KUKA KRL data list: profile_defaut.dat

&ACCESS RVP
&PARAM EDITMASK = *
DEFDAT  profile_defaut
;FOLD EXTERNAL DECLARATIONS;%{PE}%MKUKATPBASIS,%CEXT,%VCOMMON,%P
;FOLD BASISTECH EXT;%{PE}%MKUKATPBASIS,%CEXT,%VEXT,%P
EXT  BAS (BAS_COMMAND  :IN,REAL  :IN )
DECL INT SUCCESS
;ENDFOLD (BASISTECH EXT)
;FOLD USER EXT;%{E}%MKUKATPUSER,%CEXT,%VEXT,%P
;Make your modifications here

;ENDFOLD (USER EXT)
;ENDFOLD (EXTERNAL DECLARATIONS)

INT APP_GENNUMBER = 215375
INT APP_ANSWER
INT APP_OFFSET
DECL STATE_T APP_STATE

DECL PDAT PPDATP0={VEL 100,ACC 100,APO_DIST 5,APO_MODE #CDIS,GEAR_JERK 100.0,EXAX_IGN 0}
DECL FDAT FP0={TOOL_NO 2,BASE_NO 10,IPO_FRAME #BASE,POINT2[] " ",TQ_STATE FALSE}
DECL E6AXIS XP0={A1 -1000.000,A2 -90.000,A3 90.000,A4 0.000,A5 -90.000,A6 0.000,E1 0.000,E2 0.000,E3 0.000,E4 0.000,E5 0.000,E6 0.000}

; Data for Routine_0
DECL LDAT LCPDATP1={VEL 0.1,ACC 100,APO_DIST 5,APO_FAC 50.0,ORI_TYP #VAR,CIRC_TYP #BASE,JERK_FAC 50.0}
DECL FDAT FP1={TOOL_NO 2,BASE_NO 10,IPO_FRAME #BASE,POINT2[] " ",TQ_STATE FALSE}
DECL E6POS XP1={X -118.780,Y -0.350,Z 2.610,A -0.040,B -12.450,C -29.720}
DECL LDAT LCPDATC2={VEL 0.1,ACC 100,APO_DIST 5,APO_FAC 50.0,ORI_TYP #VAR,CIRC_TYP #BASE,JERK_FAC 50.0}
DECL FDAT FC2={TOOL_NO 2,BASE_NO 10,IPO_FRAME #BASE,POINT2[] " ",TQ_STATE FALSE}
DECL E6POS XCAux2={X -55.000,Y 13.210,Z 2.610,A 0.000,B 0.000,C -32.000}
DECL E6POS XCDes2={X 8.780,Y -0.350,Z 2.610,A 0.040,B 12.450,C -29.720}
DECL LDAT LCPDATC3={VEL 0.5,ACC 100,APO_DIST 5,APO_FAC 50.0,ORI_TYP #VAR,CIRC_TYP #BASE,JERK_FAC 50.0}
DECL FDAT FC3={TOOL_NO 2,BASE_NO 10,IPO_FRAME #BASE,POINT2[] " ",TQ_STATE FALSE}
DECL E6POS XCAux3={X 32.690,Y -13.600,Z 2.610,A 0.100,B 17.240,C -27.390}
DECL E6POS XCDes3={X 31.690,Y -15.080,Z 3.460,A 0.010,B 10.280,C -15.600}
DECL LDAT LCPDATP4={VEL 0.1,ACC 100,APO_DIST 5,APO_FAC 50.0,ORI_TYP #VAR,CIRC_TYP #BASE,JERK_FAC 50.0}
DECL FDAT FP4={TOOL_NO 2,BASE_NO 10,IPO_FRAME #BASE,POINT2[] " ",TQ_STATE FALSE}
DECL E6POS XP4={X 8.050,Y -1.980,Z 3.460,A 0.000,B 7.460,C -17.100}
DECL LDAT LCPDATC5={VEL 0.1,ACC 100,APO_DIST 5,APO_FAC 50.0,ORI_TYP #VAR,CIRC_TYP #BASE,JERK_FAC 50.0}
DECL FDAT FC5={TOOL_NO 2,BASE_NO 10,IPO_FRAME #BASE,POINT2[] " ",TQ_STATE FALSE}
DECL E6POS XCAux5={X -55.000,Y 11.430,Z 3.460,A 0.000,B 0.000,C -18.620}
DECL E6POS XCDes5={X -118.050,Y -1.980,Z 3.460,A -0.000,B -7.460,C -17.100}
DECL LDAT LCPDATC6={VEL 0.5,ACC 100,APO_DIST 5,APO_FAC 50.0,ORI_TYP #VAR,CIRC_TYP #BASE,JERK_FAC 50.0}
DECL FDAT FC6={TOOL_NO 2,BASE_NO 10,IPO_FRAME #BASE,POINT2[] " ",TQ_STATE FALSE}
DECL E6POS XCAux6={X -141.690,Y -15.080,Z 3.460,A -0.010,B -10.280,C -15.600}
DECL E6POS XCDes6={X -140.610,Y -16.680,Z 3.860,A -0.000,B -2.920,C -4.340}
DECL LDAT LCPDATP7={VEL 0.1,ACC 100,APO_DIST 5,APO_FAC 50.0,ORI_TYP #VAR,CIRC_TYP #BASE,JERK_FAC 50.0}
DECL FDAT FP7={TOOL_NO 2,BASE_NO 10,IPO_FRAME #BASE,POINT2[] " ",TQ_STATE FALSE}
DECL E6POS XP7={X -117.270,Y -3.740,Z 3.860,A -0.000,B -2.130,C -4.780}
DECL LDAT LCPDATC8={VEL 0.1,ACC 100,APO_DIST 5,APO_FAC 50.0,ORI_TYP #VAR,CIRC_TYP #BASE,JERK_FAC 50.0}
DECL FDAT FC8={TOOL_NO 2,BASE_NO 10,IPO_FRAME #BASE,POINT2[] " ",TQ_STATE FALSE}
DECL E6POS XCAux8={X -55.000,Y 9.500,Z 3.860,A 0.000,B 0.000,C -5.230}
DECL E6POS XCDes8={X 7.270,Y -3.740,Z 3.860,A 0.000,B 2.130,C -4.780}
DECL LDAT LCPDATC9={VEL 0.5,ACC 100,APO_DIST 5,APO_FAC 50.0,ORI_TYP #VAR,CIRC_TYP #BASE,JERK_FAC 50.0}
DECL FDAT FC9={TOOL_NO 2,BASE_NO 10,IPO_FRAME #BASE,POINT2[] " ",TQ_STATE FALSE}
DECL E6POS XCAux9={X 30.610,Y -16.680,Z 3.860,A 0.000,B 2.920,C -4.340}
DECL E6POS XCDes9={X 30.620,Y -16.670,Z 3.900,A 0.000,B 0.000,C -0.000}
DECL LDAT LCPDATP10={VEL 0.1,ACC 100,APO_DIST 5,APO_FAC 50.0,ORI_TYP #VAR,CIRC_TYP #BASE,JERK_FAC 50.0}
DECL FDAT FP10={TOOL_NO 2,BASE_NO 10,IPO_FRAME #BASE,POINT2[] " ",TQ_STATE FALSE}
DECL E6POS XP10={X 7.270,Y -3.730,Z 3.900,A 0.000,B 0.000,C -0.000}
DECL LDAT LCPDATC11={VEL 0.1,ACC 100,APO_DIST 5,APO_FAC 50.0,ORI_TYP #VAR,CIRC_TYP #BASE,JERK_FAC 50.0}
DECL FDAT FC11={TOOL_NO 2,BASE_NO 10,IPO_FRAME #BASE,POINT2[] " ",TQ_STATE FALSE}
DECL E6POS XCAux11={X -55.000,Y 9.510,Z 3.900,A 0.000,B 0.000,C -0.000}
DECL E6POS XCDes11={X -117.270,Y -3.730,Z 3.900,A 0.000,B 0.000,C -0.000}
DECL LDAT LCPDATC12={VEL 0.5,ACC 100,APO_DIST 5,APO_FAC 50.0,ORI_TYP #VAR,CIRC_TYP #BASE,JERK_FAC 50.0}
DECL FDAT FC12={TOOL_NO 2,BASE_NO 10,IPO_FRAME #BASE,POINT2[] " ",TQ_STATE FALSE}
DECL E6POS XCAux12={X -140.620,Y -16.670,Z 3.900,A 0.000,B 0.000,C -0.000}
DECL E6POS XCDes12={X -139.500,Y -18.330,Z 3.900,A 0.000,B 0.000,C -0.000}
DECL LDAT LCPDATP13={VEL 0.1,ACC 100,APO_DIST 5,APO_FAC 50.0,ORI_TYP #VAR,CIRC_TYP #BASE,JERK_FAC 50.0}
DECL FDAT FP13={TOOL_NO 2,BASE_NO 10,IPO_FRAME #BASE,POINT2[] " ",TQ_STATE FALSE}
DECL E6POS XP13={X -116.460,Y -5.560,Z 3.900,A 0.000,B 0.000,C -0.000}
DECL LDAT LCPDATC14={VEL 0.1,ACC 100,APO_DIST 5,APO_FAC 50.0,ORI_TYP #VAR,CIRC_TYP #BASE,JERK_FAC 50.0}
DECL FDAT FC14={TOOL_NO 2,BASE_NO 10,IPO_FRAME #BASE,POINT2[] " ",TQ_STATE FALSE}
DECL E6POS XCAux14={X -55.000,Y 7.510,Z 3.900,A 0.000,B 0.000,C -0.000}
DECL E6POS XCDes14={X 6.460,Y -5.560,Z 3.900,A 0.000,B 0.000,C -0.000}
DECL LDAT LCPDATC15={VEL 0.5,ACC 100,APO_DIST 5,APO_FAC 50.0,ORI_TYP #VAR,CIRC_TYP #BASE,JERK_FAC 50.0}
DECL FDAT FC15={TOOL_NO 2,BASE_NO 10,IPO_FRAME #BASE,POINT2[] " ",TQ_STATE FALSE}
DECL E6POS XCAux15={X 29.500,Y -18.330,Z 3.900,A 0.000,B 0.000,C -0.000}
DECL E6POS XCDes15={X 28.380,Y -19.990,Z 3.900,A 0.000,B 0.000,C -0.000}
DECL LDAT LCPDATP16={VEL 0.1,ACC 100,APO_DIST 5,APO_FAC 50.0,ORI_TYP #VAR,CIRC_TYP #BASE,JERK_FAC 50.0}
DECL FDAT FP16={TOOL_NO 2,BASE_NO 10,IPO_FRAME #BASE,POINT2[] " ",TQ_STATE FALSE}
DECL E6POS XP16={X 5.650,Y -7.390,Z 3.900,A 0.000,B 0.000,C -0.000}
DECL LDAT LCPDATC17={VEL 0.1,ACC 100,APO_DIST 5,APO_FAC 50.0,ORI_TYP #VAR,CIRC_TYP #BASE,JERK_FAC 50.0}
DECL FDAT FC17={TOOL_NO 2,BASE_NO 10,IPO_FRAME #BASE,POINT2[] " ",TQ_STATE FALSE}
DECL E6POS XCAux17={X -55.000,Y 5.510,Z 3.900,A 0.000,B 0.000,C -0.000}
DECL E6POS XCDes17={X -115.650,Y -7.390,Z 3.900,A 0.000,B 0.000,C -0.000}
DECL LDAT LCPDATC18={VEL 0.5,ACC 100,APO_DIST 5,APO_FAC 50.0,ORI_TYP #VAR,CIRC_TYP #BASE,JERK_FAC 50.0}
DECL FDAT FC18={TOOL_NO 2,BASE_NO 10,IPO_FRAME #BASE,POINT2[] " ",TQ_STATE FALSE}
DECL E6POS XCAux18={X -138.380,Y -19.990,Z 3.900,A 0.000,B 0.000,C -0.000}
DECL E6POS XCDes18={X -137.260,Y -21.640,Z 3.900,A 0.000,B 0.000,C -0.000}
DECL LDAT LCPDATP19={VEL 0.1,ACC 100,APO_DIST 5,APO_FAC 50.0,ORI_TYP #VAR,CIRC_TYP #BASE,JERK_FAC 50.0}
DECL FDAT FP19={TOOL_NO 2,BASE_NO 10,IPO_FRAME #BASE,POINT2[] " ",TQ_STATE FALSE}
DECL E6POS XP19={X -114.830,Y -9.210,Z 3.900,A 0.000,B 0.000,C -0.000}
DECL LDAT LCPDATC20={VEL 0.1,ACC 100,APO_DIST 5,APO_FAC 50.0,ORI_TYP #VAR,CIRC_TYP #BASE,JERK_FAC 50.0}
DECL FDAT FC20={TOOL_NO 2,BASE_NO 10,IPO_FRAME #BASE,POINT2[] " ",TQ_STATE FALSE}
DECL E6POS XCAux20={X -55.000,Y 3.510,Z 3.900,A 0.000,B 0.000,C -0.000}
DECL E6POS XCDes20={X 4.830,Y -9.210,Z 3.900,A 0.000,B 0.000,C -0.000}
DECL LDAT LCPDATC21={VEL 0.5,ACC 100,APO_DIST 5,APO_FAC 50.0,ORI_TYP #VAR,CIRC_TYP #BASE,JERK_FAC 50.0}
DECL FDAT FC21={TOOL_NO 2,BASE_NO 10,IPO_FRAME #BASE,POINT2[] " ",TQ_STATE FALSE}
DECL E6POS XCAux21={X 27.260,Y -21.640,Z 3.900,A 0.000,B 0.000,C -0.000}
DECL E6POS XCDes21={X 26.140,Y -23.300,Z 3.900,A 0.000,B 0.000,C -0.000}
DECL LDAT LCPDATP22={VEL 0.1,ACC 100,APO_DIST 5,APO_FAC 50.0,ORI_TYP #VAR,CIRC_TYP #BASE,JERK_FAC 50.0}
DECL FDAT FP22={TOOL_NO 2,BASE_NO 10,IPO_FRAME #BASE,POINT2[] " ",TQ_STATE FALSE}
DECL E6POS XP22={X 4.020,Y -11.040,Z 3.900,A 0.000,B 0.000,C -0.000}
DECL LDAT LCPDATC23={VEL 0.1,ACC 100,APO_DIST 5,APO_FAC 50.0,ORI_TYP #VAR,CIRC_TYP #BASE,JERK_FAC 50.0}
DECL FDAT FC23={TOOL_NO 2,BASE_NO 10,IPO_FRAME #BASE,POINT2[] " ",TQ_STATE FALSE}
DECL E6POS XCAux23={X -55.000,Y 1.510,Z 3.900,A 0.000,B 0.000,C -0.000}
DECL E6POS XCDes23={X -114.020,Y -11.040,Z 3.900,A 0.000,B 0.000,C -0.000}
DECL LDAT LCPDATC24={VEL 0.5,ACC 100,APO_DIST 5,APO_FAC 50.0,ORI_TYP #VAR,CIRC_TYP #BASE,JERK_FAC 50.0}
DECL FDAT FC24={TOOL_NO 2,BASE_NO 10,IPO_FRAME #BASE,POINT2[] " ",TQ_STATE FALSE}
DECL E6POS XCAux24={X -136.140,Y -23.300,Z 3.900,A 0.000,B 0.000,C -0.000}
DECL E6POS XCDes24={X -135.020,Y -24.960,Z 3.900,A 0.000,B 0.000,C -0.000}
DECL LDAT LCPDATP25={VEL 0.1,ACC 100,APO_DIST 5,APO_FAC 50.0,ORI_TYP #VAR,CIRC_TYP #BASE,JERK_FAC 50.0}
DECL FDAT FP25={TOOL_NO 2,BASE_NO 10,IPO_FRAME #BASE,POINT2[] " ",TQ_STATE FALSE}
DECL E6POS XP25={X -113.210,Y -12.870,Z 3.900,A 0.000,B 0.000,C -0.000}
DECL LDAT LCPDATC26={VEL 0.1,ACC 100,APO_DIST 5,APO_FAC 50.0,ORI_TYP #VAR,CIRC_TYP #BASE,JERK_FAC 50.0}
DECL FDAT FC26={TOOL_NO 2,BASE_NO 10,IPO_FRAME #BASE,POINT2[] " ",TQ_STATE FALSE}
DECL E6POS XCAux26={X -55.000,Y -0.490,Z 3.900,A 0.000,B 0.000,C -0.000}
DECL E6POS XCDes26={X 3.210,Y -12.870,Z 3.900,A 0.000,B 0.000,C -0.000}
DECL LDAT LCPDATC27={VEL 0.5,ACC 100,APO_DIST 5,APO_FAC 50.0,ORI_TYP #VAR,CIRC_TYP #BASE,JERK_FAC 50.0}
DECL FDAT FC27={TOOL_NO 2,BASE_NO 10,IPO_FRAME #BASE,POINT2[] " ",TQ_STATE FALSE}
DECL E6POS XCAux27={X 25.020,Y -24.960,Z 3.900,A 0.000,B 0.000,C -0.000}
DECL E6POS XCDes27={X 23.910,Y -26.620,Z 3.900,A 0.000,B 0.000,C -0.000}
DECL LDAT LCPDATP28={VEL 0.1,ACC 100,APO_DIST 5,APO_FAC 50.0,ORI_TYP #VAR,CIRC_TYP #BASE,JERK_FAC 50.0}
DECL FDAT FP28={TOOL_NO 2,BASE_NO 10,IPO_FRAME #BASE,POINT2[] " ",TQ_STATE FALSE}
DECL E6POS XP28={X 2.390,Y -14.690,Z 3.900,A 0.000,B 0.000,C -0.000}
DECL LDAT LCPDATC29={VEL 0.1,ACC 100,APO_DIST 5,APO_FAC 50.0,ORI_TYP #VAR,CIRC_TYP #BASE,JERK_FAC 50.0}
DECL FDAT FC29={TOOL_NO 2,BASE_NO 10,IPO_FRAME #BASE,POINT2[] " ",TQ_STATE FALSE}
DECL E6POS XCAux29={X -55.000,Y -2.490,Z 3.900,A 0.000,B 0.000,C -0.000}
DECL E6POS XCDes29={X -112.390,Y -14.690,Z 3.900,A 0.000,B 0.000,C -0.000}
DECL LDAT LCPDATC30={VEL 0.5,ACC 100,APO_DIST 5,APO_FAC 50.0,ORI_TYP #VAR,CIRC_TYP #BASE,JERK_FAC 50.0}
DECL FDAT FC30={TOOL_NO 2,BASE_NO 10,IPO_FRAME #BASE,POINT2[] " ",TQ_STATE FALSE}
DECL E6POS XCAux30={X -133.910,Y -26.620,Z 3.900,A 0.000,B 0.000,C -0.000}
DECL E6POS XCDes30={X -132.790,Y -28.280,Z 3.900,A 0.000,B 0.000,C -0.000}
DECL LDAT LCPDATP31={VEL 0.1,ACC 100,APO_DIST 5,APO_FAC 50.0,ORI_TYP #VAR,CIRC_TYP #BASE,JERK_FAC 50.0}
DECL FDAT FP31={TOOL_NO 2,BASE_NO 10,IPO_FRAME #BASE,POINT2[] " ",TQ_STATE FALSE}
DECL E6POS XP31={X -111.580,Y -16.520,Z 3.900,A 0.000,B 0.000,C -0.000}
DECL LDAT LCPDATC32={VEL 0.1,ACC 100,APO_DIST 5,APO_FAC 50.0,ORI_TYP #VAR,CIRC_TYP #BASE,JERK_FAC 50.0}
DECL FDAT FC32={TOOL_NO 2,BASE_NO 10,IPO_FRAME #BASE,POINT2[] " ",TQ_STATE FALSE}
DECL E6POS XCAux32={X -55.000,Y -4.490,Z 3.900,A 0.000,B 0.000,C -0.000}
DECL E6POS XCDes32={X 1.580,Y -16.520,Z 3.900,A 0.000,B 0.000,C -0.000}
DECL LDAT LCPDATC33={VEL 0.5,ACC 100,APO_DIST 5,APO_FAC 50.0,ORI_TYP #VAR,CIRC_TYP #BASE,JERK_FAC 50.0}
DECL FDAT FC33={TOOL_NO 2,BASE_NO 10,IPO_FRAME #BASE,POINT2[] " ",TQ_STATE FALSE}
DECL E6POS XCAux33={X 22.790,Y -28.280,Z 3.900,A 0.000,B 0.000,C -0.000}
DECL E6POS XCDes33={X 22.000,Y -29.440,Z 3.900,A 0.000,B 0.090,C -0.140}
DECL LDAT LCPDATP34={VEL 0.1,ACC 100,APO_DIST 5,APO_FAC 50.0,ORI_TYP #VAR,CIRC_TYP #BASE,JERK_FAC 50.0}
DECL FDAT FP34={TOOL_NO 2,BASE_NO 10,IPO_FRAME #BASE,POINT2[] " ",TQ_STATE FALSE}
DECL E6POS XP34={X 1.010,Y -17.800,Z 3.900,A 0.000,B 0.070,C -0.150}
DECL LDAT LCPDATC35={VEL 0.1,ACC 100,APO_DIST 5,APO_FAC 50.0,ORI_TYP #VAR,CIRC_TYP #BASE,JERK_FAC 50.0}
DECL FDAT FC35={TOOL_NO 2,BASE_NO 10,IPO_FRAME #BASE,POINT2[] " ",TQ_STATE FALSE}
DECL E6POS XCAux35={X -55.000,Y -5.900,Z 3.900,A 0.000,B 0.000,C -0.170}
DECL E6POS XCDes35={X -111.010,Y -17.800,Z 3.900,A -0.000,B -0.070,C -0.150}
DECL LDAT LCPDATC36={VEL 0.5,ACC 100,APO_DIST 5,APO_FAC 50.0,ORI_TYP #VAR,CIRC_TYP #BASE,JERK_FAC 50.0}
DECL FDAT FC36={TOOL_NO 2,BASE_NO 10,IPO_FRAME #BASE,POINT2[] " ",TQ_STATE FALSE}
DECL E6POS XCAux36={X -132.000,Y -29.440,Z 3.900,A -0.000,B -0.090,C -0.140}
DECL E6POS XCDes36={X -130.910,Y -31.070,Z 3.680,A -0.000,B 7.350,C 11.020}
DECL LDAT LCPDATP37={VEL 0.1,ACC 100,APO_DIST 5,APO_FAC 50.0,ORI_TYP #VAR,CIRC_TYP #BASE,JERK_FAC 50.0}
DECL FDAT FP37={TOOL_NO 2,BASE_NO 10,IPO_FRAME #BASE,POINT2[] " ",TQ_STATE FALSE}
DECL E6POS XP37={X -110.210,Y -19.590,Z 3.680,A -0.000,B 5.340,C 12.110}
DECL LDAT LCPDATC38={VEL 0.1,ACC 100,APO_DIST 5,APO_FAC 50.0,ORI_TYP #VAR,CIRC_TYP #BASE,JERK_FAC 50.0}
DECL FDAT FC38={TOOL_NO 2,BASE_NO 10,IPO_FRAME #BASE,POINT2[] " ",TQ_STATE FALSE}
DECL E6POS XCAux38={X -55.000,Y -7.860,Z 3.680,A 0.000,B 0.000,C 13.220}
DECL E6POS XCDes38={X 0.210,Y -19.590,Z 3.680,A 0.000,B -5.340,C 12.110}
DECL LDAT LCPDATC39={VEL 0.5,ACC 100,APO_DIST 5,APO_FAC 50.0,ORI_TYP #VAR,CIRC_TYP #BASE,JERK_FAC 50.0}
DECL FDAT FC39={TOOL_NO 2,BASE_NO 10,IPO_FRAME #BASE,POINT2[] " ",TQ_STATE FALSE}
DECL E6POS XCAux39={X 20.910,Y -31.070,Z 3.680,A 0.000,B -7.350,C 11.020}
DECL E6POS XCDes39={X 19.870,Y -32.600,Z 3.000,A 0.050,B -14.500,C 22.550}
DECL LDAT LCPDATP40={VEL 0.1,ACC 100,APO_DIST 5,APO_FAC 50.0,ORI_TYP #VAR,CIRC_TYP #BASE,JERK_FAC 50.0}
DECL FDAT FP40={TOOL_NO 2,BASE_NO 10,IPO_FRAME #BASE,POINT2[] " ",TQ_STATE FALSE}
DECL E6POS XP40={X -0.540,Y -21.290,Z 3.000,A 0.020,B -10.490,C 24.580}
DECL LDAT LCPDATC41={VEL 0.1,ACC 100,APO_DIST 5,APO_FAC 50.0,ORI_TYP #VAR,CIRC_TYP #BASE,JERK_FAC 50.0}
DECL FDAT FC41={TOOL_NO 2,BASE_NO 10,IPO_FRAME #BASE,POINT2[] " ",TQ_STATE FALSE}
DECL E6POS XCAux41={X -55.000,Y -9.710,Z 3.000,A 0.000,B 0.000,C 26.600}
DECL E6POS XCDes41={X -109.460,Y -21.290,Z 3.000,A -0.020,B 10.490,C 24.580}
DECL LDAT LCPDATC42={VEL 0.5,ACC 100,APO_DIST 5,APO_FAC 50.0,ORI_TYP #VAR,CIRC_TYP #BASE,JERK_FAC 50.0}
DECL FDAT FC42={TOOL_NO 2,BASE_NO 10,IPO_FRAME #BASE,POINT2[] " ",TQ_STATE FALSE}
DECL E6POS XCAux42={X -129.870,Y -32.600,Z 3.000,A -0.050,B 14.500,C 22.550}
DECL E6POS XCDes42={X -129.880,Y -32.590,Z 2.560,A -0.060,B 15.190,C 23.730}
DECL LDAT LCPDATP43={VEL 0.1,ACC 100,APO_DIST 5,APO_FAC 50.0,ORI_TYP #VAR,CIRC_TYP #BASE,JERK_FAC 50.0}
DECL FDAT FP43={TOOL_NO 2,BASE_NO 10,IPO_FRAME #BASE,POINT2[] " ",TQ_STATE FALSE}
DECL E6POS XP43={X -109.460,Y -21.280,Z 2.560,A -0.020,B 10.980,C 25.840}
DECL LDAT LCPDATC44={VEL 0.1,ACC 100,APO_DIST 5,APO_FAC 50.0,ORI_TYP #VAR,CIRC_TYP #BASE,JERK_FAC 50.0}
DECL FDAT FC44={TOOL_NO 2,BASE_NO 10,IPO_FRAME #BASE,POINT2[] " ",TQ_STATE FALSE}
DECL E6POS XCAux44={X -55.000,Y -9.700,Z 2.560,A 0.000,B 0.000,C 27.930}
DECL E6POS XCDes44={X -0.540,Y -21.280,Z 2.560,A 0.020,B -10.980,C 25.840}
DECL LDAT LCPDATC45={VEL 0.5,ACC 100,APO_DIST 5,APO_FAC 50.0,ORI_TYP #VAR,CIRC_TYP #BASE,JERK_FAC 50.0}
DECL FDAT FC45={TOOL_NO 2,BASE_NO 10,IPO_FRAME #BASE,POINT2[] " ",TQ_STATE FALSE}
DECL E6POS XCAux45={X 19.880,Y -32.590,Z 2.560,A 0.060,B -15.190,C 23.730}
DECL E6POS XCDes45={X 20.900,Y -31.070,Z 3.260,A 0.000,B -7.720,C 11.590}
DECL LDAT LCPDATP46={VEL 0.1,ACC 100,APO_DIST 5,APO_FAC 50.0,ORI_TYP #VAR,CIRC_TYP #BASE,JERK_FAC 50.0}
DECL FDAT FP46={TOOL_NO 2,BASE_NO 10,IPO_FRAME #BASE,POINT2[] " ",TQ_STATE FALSE}
DECL E6POS XP46={X 0.210,Y -19.600,Z 3.260,A 0.000,B -5.600,C 12.730}
DECL LDAT LCPDATC47={VEL 0.1,ACC 100,APO_DIST 5,APO_FAC 50.0,ORI_TYP #VAR,CIRC_TYP #BASE,JERK_FAC 50.0}
DECL FDAT FC47={TOOL_NO 2,BASE_NO 10,IPO_FRAME #BASE,POINT2[] " ",TQ_STATE FALSE}
DECL E6POS XCAux47={X -55.000,Y -7.860,Z 3.260,A 0.000,B 0.000,C 13.890}
DECL E6POS XCDes47={X -110.210,Y -19.600,Z 3.260,A -0.000,B 5.600,C 12.730}
DECL LDAT LCPDATC48={VEL 0.5,ACC 100,APO_DIST 5,APO_FAC 50.0,ORI_TYP #VAR,CIRC_TYP #BASE,JERK_FAC 50.0}
DECL FDAT FC48={TOOL_NO 2,BASE_NO 10,IPO_FRAME #BASE,POINT2[] " ",TQ_STATE FALSE}
DECL E6POS XCAux48={X -130.900,Y -31.070,Z 3.260,A -0.000,B 7.720,C 11.590}
DECL E6POS XCDes48={X -132.000,Y -29.440,Z 3.500,A -0.000,B -0.080,C -0.120}
DECL LDAT LCPDATP49={VEL 0.1,ACC 100,APO_DIST 5,APO_FAC 50.0,ORI_TYP #VAR,CIRC_TYP #BASE,JERK_FAC 50.0}
DECL FDAT FP49={TOOL_NO 2,BASE_NO 10,IPO_FRAME #BASE,POINT2[] " ",TQ_STATE FALSE}
DECL E6POS XP49={X -111.010,Y -17.810,Z 3.500,A -0.000,B -0.060,C -0.140}
DECL LDAT LCPDATC50={VEL 0.1,ACC 100,APO_DIST 5,APO_FAC 50.0,ORI_TYP #VAR,CIRC_TYP #BASE,JERK_FAC 50.0}
DECL FDAT FC50={TOOL_NO 2,BASE_NO 10,IPO_FRAME #BASE,POINT2[] " ",TQ_STATE FALSE}
DECL E6POS XCAux50={X -55.000,Y -5.900,Z 3.500,A 0.000,B 0.000,C -0.150}
DECL E6POS XCDes50={X 1.010,Y -17.810,Z 3.500,A 0.000,B 0.060,C -0.140}
DECL LDAT LCPDATC51={VEL 0.5,ACC 100,APO_DIST 5,APO_FAC 50.0,ORI_TYP #VAR,CIRC_TYP #BASE,JERK_FAC 50.0}
DECL FDAT FC51={TOOL_NO 2,BASE_NO 10,IPO_FRAME #BASE,POINT2[] " ",TQ_STATE FALSE}
DECL E6POS XCAux51={X 22.000,Y -29.440,Z 3.500,A 0.000,B 0.080,C -0.120}
DECL E6POS XCDes51={X 22.660,Y -28.460,Z 3.500,A 0.000,B 0.000,C -0.000}
DECL LDAT LCPDATP52={VEL 0.1,ACC 100,APO_DIST 5,APO_FAC 50.0,ORI_TYP #VAR,CIRC_TYP #BASE,JERK_FAC 50.0}
DECL FDAT FP52={TOOL_NO 2,BASE_NO 10,IPO_FRAME #BASE,POINT2[] " ",TQ_STATE FALSE}
DECL E6POS XP52={X 1.490,Y -16.720,Z 3.500,A 0.000,B 0.000,C -0.000}
DECL LDAT LCPDATC53={VEL 0.1,ACC 100,APO_DIST 5,APO_FAC 50.0,ORI_TYP #VAR,CIRC_TYP #BASE,JERK_FAC 50.0}
DECL FDAT FC53={TOOL_NO 2,BASE_NO 10,IPO_FRAME #BASE,POINT2[] " ",TQ_STATE FALSE}
DECL E6POS XCAux53={X -55.000,Y -4.720,Z 3.500,A 0.000,B 0.000,C -0.000}
DECL E6POS XCDes53={X -111.490,Y -16.720,Z 3.500,A 0.000,B 0.000,C -0.000}
DECL LDAT LCPDATC54={VEL 0.5,ACC 100,APO_DIST 5,APO_FAC 50.0,ORI_TYP #VAR,CIRC_TYP #BASE,JERK_FAC 50.0}
DECL FDAT FC54={TOOL_NO 2,BASE_NO 10,IPO_FRAME #BASE,POINT2[] " ",TQ_STATE FALSE}
DECL E6POS XCAux54={X -132.660,Y -28.460,Z 3.500,A 0.000,B 0.000,C -0.000}
DECL E6POS XCDes54={X -133.780,Y -26.800,Z 3.500,A 0.000,B 0.000,C -0.000}
DECL LDAT LCPDATP55={VEL 0.1,ACC 100,APO_DIST 5,APO_FAC 50.0,ORI_TYP #VAR,CIRC_TYP #BASE,JERK_FAC 50.0}
DECL FDAT FP55={TOOL_NO 2,BASE_NO 10,IPO_FRAME #BASE,POINT2[] " ",TQ_STATE FALSE}
DECL E6POS XP55={X -112.300,Y -14.900,Z 3.500,A 0.000,B 0.000,C -0.000}
DECL LDAT LCPDATC56={VEL 0.1,ACC 100,APO_DIST 5,APO_FAC 50.0,ORI_TYP #VAR,CIRC_TYP #BASE,JERK_FAC 50.0}
DECL FDAT FC56={TOOL_NO 2,BASE_NO 10,IPO_FRAME #BASE,POINT2[] " ",TQ_STATE FALSE}
DECL E6POS XCAux56={X -55.000,Y -2.720,Z 3.500,A 0.000,B 0.000,C -0.000}
DECL E6POS XCDes56={X 2.300,Y -14.900,Z 3.500,A 0.000,B 0.000,C -0.000}
DECL LDAT LCPDATC57={VEL 0.5,ACC 100,APO_DIST 5,APO_FAC 50.0,ORI_TYP #VAR,CIRC_TYP #BASE,JERK_FAC 50.0}
DECL FDAT FC57={TOOL_NO 2,BASE_NO 10,IPO_FRAME #BASE,POINT2[] " ",TQ_STATE FALSE}
DECL E6POS XCAux57={X 23.780,Y -26.800,Z 3.500,A 0.000,B 0.000,C -0.000}
DECL E6POS XCDes57={X 24.900,Y -25.140,Z 3.500,A 0.000,B 0.000,C -0.000}
DECL LDAT LCPDATP58={VEL 0.1,ACC 100,APO_DIST 5,APO_FAC 50.0,ORI_TYP #VAR,CIRC_TYP #BASE,JERK_FAC 50.0}
DECL FDAT FP58={TOOL_NO 2,BASE_NO 10,IPO_FRAME #BASE,POINT2[] " ",TQ_STATE FALSE}
DECL E6POS XP58={X 3.120,Y -13.070,Z 3.500,A 0.000,B 0.000,C -0.000}
DECL LDAT LCPDATC59={VEL 0.1,ACC 100,APO_DIST 5,APO_FAC 50.0,ORI_TYP #VAR,CIRC_TYP #BASE,JERK_FAC 50.0}
DECL FDAT FC59={TOOL_NO 2,BASE_NO 10,IPO_FRAME #BASE,POINT2[] " ",TQ_STATE FALSE}
DECL E6POS XCAux59={X -55.000,Y -0.720,Z 3.500,A 0.000,B 0.000,C -0.000}
DECL E6POS XCDes59={X -113.120,Y -13.070,Z 3.500,A 0.000,B 0.000,C -0.000}
DECL LDAT LCPDATC60={VEL 0.5,ACC 100,APO_DIST 5,APO_FAC 50.0,ORI_TYP #VAR,CIRC_TYP #BASE,JERK_FAC 50.0}
DECL FDAT FC60={TOOL_NO 2,BASE_NO 10,IPO_FRAME #BASE,POINT2[] " ",TQ_STATE FALSE}
DECL E6POS XCAux60={X -134.900,Y -25.140,Z 3.500,A 0.000,B 0.000,C -0.000}
DECL E6POS XCDes60={X -136.020,Y -23.490,Z 3.500,A 0.000,B 0.000,C -0.000}
DECL LDAT LCPDATP61={VEL 0.1,ACC 100,APO_DIST 5,APO_FAC 50.0,ORI_TYP #VAR,CIRC_TYP #BASE,JERK_FAC 50.0}
DECL FDAT FP61={TOOL_NO 2,BASE_NO 10,IPO_FRAME #BASE,POINT2[] " ",TQ_STATE FALSE}
DECL E6POS XP61={X -113.930,Y -11.240,Z 3.500,A 0.000,B 0.000,C -0.000}
DECL LDAT LCPDATC62={VEL 0.1,ACC 100,APO_DIST 5,APO_FAC 50.0,ORI_TYP #VAR,CIRC_TYP #BASE,JERK_FAC 50.0}
DECL FDAT FC62={TOOL_NO 2,BASE_NO 10,IPO_FRAME #BASE,POINT2[] " ",TQ_STATE FALSE}
DECL E6POS XCAux62={X -55.000,Y 1.280,Z 3.500,A 0.000,B 0.000,C -0.000}
DECL E6POS XCDes62={X 3.930,Y -11.240,Z 3.500,A 0.000,B 0.000,C -0.000}
DECL LDAT LCPDATC63={VEL 0.5,ACC 100,APO_DIST 5,APO_FAC 50.0,ORI_TYP #VAR,CIRC_TYP #BASE,JERK_FAC 50.0}
DECL FDAT FC63={TOOL_NO 2,BASE_NO 10,IPO_FRAME #BASE,POINT2[] " ",TQ_STATE FALSE}
DECL E6POS XCAux63={X 26.020,Y -23.490,Z 3.500,A 0.000,B 0.000,C -0.000}
DECL E6POS XCDes63={X 27.140,Y -21.830,Z 3.500,A 0.000,B 0.000,C -0.000}
DECL LDAT LCPDATP64={VEL 0.1,ACC 100,APO_DIST 5,APO_FAC 50.0,ORI_TYP #VAR,CIRC_TYP #BASE,JERK_FAC 50.0}
DECL FDAT FP64={TOOL_NO 2,BASE_NO 10,IPO_FRAME #BASE,POINT2[] " ",TQ_STATE FALSE}
DECL E6POS XP64={X 4.740,Y -9.420,Z 3.500,A 0.000,B 0.000,C -0.000}
DECL LDAT LCPDATC65={VEL 0.1,ACC 100,APO_DIST 5,APO_FAC 50.0,ORI_TYP #VAR,CIRC_TYP #BASE,JERK_FAC 50.0}
DECL FDAT FC65={TOOL_NO 2,BASE_NO 10,IPO_FRAME #BASE,POINT2[] " ",TQ_STATE FALSE}
DECL E6POS XCAux65={X -55.000,Y 3.280,Z 3.500,A 0.000,B 0.000,C -0.000}
DECL E6POS XCDes65={X -114.740,Y -9.420,Z 3.500,A 0.000,B 0.000,C -0.000}
DECL LDAT LCPDATC66={VEL 0.5,ACC 100,APO_DIST 5,APO_FAC 50.0,ORI_TYP #VAR,CIRC_TYP #BASE,JERK_FAC 50.0}
DECL FDAT FC66={TOOL_NO 2,BASE_NO 10,IPO_FRAME #BASE,POINT2[] " ",TQ_STATE FALSE}
DECL E6POS XCAux66={X -137.140,Y -21.830,Z 3.500,A 0.000,B 0.000,C -0.000}
DECL E6POS XCDes66={X -138.250,Y -20.170,Z 3.500,A 0.000,B 0.000,C -0.000}
DECL LDAT LCPDATP67={VEL 0.1,ACC 100,APO_DIST 5,APO_FAC 50.0,ORI_TYP #VAR,CIRC_TYP #BASE,JERK_FAC 50.0}
DECL FDAT FP67={TOOL_NO 2,BASE_NO 10,IPO_FRAME #BASE,POINT2[] " ",TQ_STATE FALSE}
DECL E6POS XP67={X -115.560,Y -7.590,Z 3.500,A 0.000,B 0.000,C -0.000}
DECL LDAT LCPDATC68={VEL 0.1,ACC 100,APO_DIST 5,APO_FAC 50.0,ORI_TYP #VAR,CIRC_TYP #BASE,JERK_FAC 50.0}
DECL FDAT FC68={TOOL_NO 2,BASE_NO 10,IPO_FRAME #BASE,POINT2[] " ",TQ_STATE FALSE}
DECL E6POS XCAux68={X -55.000,Y 5.280,Z 3.500,A 0.000,B 0.000,C -0.000}
DECL E6POS XCDes68={X 5.560,Y -7.590,Z 3.500,A 0.000,B 0.000,C -0.000}
DECL LDAT LCPDATC69={VEL 0.5,ACC 100,APO_DIST 5,APO_FAC 50.0,ORI_TYP #VAR,CIRC_TYP #BASE,JERK_FAC 50.0}
DECL FDAT FC69={TOOL_NO 2,BASE_NO 10,IPO_FRAME #BASE,POINT2[] " ",TQ_STATE FALSE}
DECL E6POS XCAux69={X 28.250,Y -20.170,Z 3.500,A 0.000,B 0.000,C -0.000}
DECL E6POS XCDes69={X 29.370,Y -18.510,Z 3.500,A 0.000,B 0.000,C -0.000}
DECL LDAT LCPDATP70={VEL 0.1,ACC 100,APO_DIST 5,APO_FAC 50.0,ORI_TYP #VAR,CIRC_TYP #BASE,JERK_FAC 50.0}
DECL FDAT FP70={TOOL_NO 2,BASE_NO 10,IPO_FRAME #BASE,POINT2[] " ",TQ_STATE FALSE}
DECL E6POS XP70={X 6.370,Y -5.760,Z 3.500,A 0.000,B 0.000,C -0.000}
DECL LDAT LCPDATC71={VEL 0.1,ACC 100,APO_DIST 5,APO_FAC 50.0,ORI_TYP #VAR,CIRC_TYP #BASE,JERK_FAC 50.0}
DECL FDAT FC71={TOOL_NO 2,BASE_NO 10,IPO_FRAME #BASE,POINT2[] " ",TQ_STATE FALSE}
DECL E6POS XCAux71={X -55.000,Y 7.280,Z 3.500,A 0.000,B 0.000,C -0.000}
DECL E6POS XCDes71={X -116.370,Y -5.760,Z 3.500,A 0.000,B 0.000,C -0.000}
DECL LDAT LCPDATC72={VEL 0.5,ACC 100,APO_DIST 5,APO_FAC 50.0,ORI_TYP #VAR,CIRC_TYP #BASE,JERK_FAC 50.0}
DECL FDAT FC72={TOOL_NO 2,BASE_NO 10,IPO_FRAME #BASE,POINT2[] " ",TQ_STATE FALSE}
DECL E6POS XCAux72={X -139.370,Y -18.510,Z 3.500,A 0.000,B 0.000,C -0.000}
DECL E6POS XCDes72={X -140.490,Y -16.850,Z 3.500,A 0.000,B 0.000,C -0.000}
DECL LDAT LCPDATP73={VEL 0.1,ACC 100,APO_DIST 5,APO_FAC 50.0,ORI_TYP #VAR,CIRC_TYP #BASE,JERK_FAC 50.0}
DECL FDAT FP73={TOOL_NO 2,BASE_NO 10,IPO_FRAME #BASE,POINT2[] " ",TQ_STATE FALSE}
DECL E6POS XP73={X -117.180,Y -3.930,Z 3.500,A 0.000,B 0.000,C -0.000}
DECL LDAT LCPDATC74={VEL 0.1,ACC 100,APO_DIST 5,APO_FAC 50.0,ORI_TYP #VAR,CIRC_TYP #BASE,JERK_FAC 50.0}
DECL FDAT FC74={TOOL_NO 2,BASE_NO 10,IPO_FRAME #BASE,POINT2[] " ",TQ_STATE FALSE}
DECL E6POS XCAux74={X -55.000,Y 9.280,Z 3.500,A 0.000,B 0.000,C -0.000}
DECL E6POS XCDes74={X 7.180,Y -3.930,Z 3.500,A 0.000,B 0.000,C -0.000}
DECL LDAT LCPDATC75={VEL 0.5,ACC 100,APO_DIST 5,APO_FAC 50.0,ORI_TYP #VAR,CIRC_TYP #BASE,JERK_FAC 50.0}
DECL FDAT FC75={TOOL_NO 2,BASE_NO 10,IPO_FRAME #BASE,POINT2[] " ",TQ_STATE FALSE}
DECL E6POS XCAux75={X 30.490,Y -16.850,Z 3.500,A 0.000,B 0.000,C -0.000}
DECL E6POS XCDes75={X 30.490,Y -16.860,Z 3.480,A 0.000,B 2.190,C -3.250}
DECL LDAT LCPDATP76={VEL 0.1,ACC 100,APO_DIST 5,APO_FAC 50.0,ORI_TYP #VAR,CIRC_TYP #BASE,JERK_FAC 50.0}
DECL FDAT FP76={TOOL_NO 2,BASE_NO 10,IPO_FRAME #BASE,POINT2[] " ",TQ_STATE FALSE}
DECL E6POS XP76={X 7.180,Y -3.940,Z 3.480,A 0.000,B 1.590,C -3.580}
DECL LDAT LCPDATC77={VEL 0.1,ACC 100,APO_DIST 5,APO_FAC 50.0,ORI_TYP #VAR,CIRC_TYP #BASE,JERK_FAC 50.0}
DECL FDAT FC77={TOOL_NO 2,BASE_NO 10,IPO_FRAME #BASE,POINT2[] " ",TQ_STATE FALSE}
DECL E6POS XCAux77={X -55.000,Y 9.280,Z 3.480,A 0.000,B 0.000,C -3.920}
DECL E6POS XCDes77={X -117.180,Y -3.940,Z 3.480,A -0.000,B -1.590,C -3.580}
DECL LDAT LCPDATC78={VEL 0.5,ACC 100,APO_DIST 5,APO_FAC 50.0,ORI_TYP #VAR,CIRC_TYP #BASE,JERK_FAC 50.0}
DECL FDAT FC78={TOOL_NO 2,BASE_NO 10,IPO_FRAME #BASE,POINT2[] " ",TQ_STATE FALSE}
DECL E6POS XCAux78={X -140.490,Y -16.860,Z 3.480,A -0.000,B -2.190,C -3.250}
DECL E6POS XCDes78={X -141.570,Y -15.260,Z 3.110,A -0.010,B -9.930,C -15.040}
DECL LDAT LCPDATP79={VEL 0.1,ACC 100,APO_DIST 5,APO_FAC 50.0,ORI_TYP #VAR,CIRC_TYP #BASE,JERK_FAC 50.0}
DECL FDAT FP79={TOOL_NO 2,BASE_NO 10,IPO_FRAME #BASE,POINT2[] " ",TQ_STATE FALSE}
DECL E6POS XP79={X -117.970,Y -2.170,Z 3.110,A -0.000,B -7.200,C -16.490}
DECL LDAT LCPDATC80={VEL 0.1,ACC 100,APO_DIST 5,APO_FAC 50.0,ORI_TYP #VAR,CIRC_TYP #BASE,JERK_FAC 50.0}
DECL FDAT FC80={TOOL_NO 2,BASE_NO 10,IPO_FRAME #BASE,POINT2[] " ",TQ_STATE FALSE}
DECL E6POS XCAux80={X -55.000,Y 11.210,Z 3.110,A 0.000,B 0.000,C -17.960}
DECL E6POS XCDes80={X 7.970,Y -2.170,Z 3.110,A 0.000,B 7.200,C -16.490}
DECL LDAT LCPDATC81={VEL 0.5,ACC 100,APO_DIST 5,APO_FAC 50.0,ORI_TYP #VAR,CIRC_TYP #BASE,JERK_FAC 50.0}
DECL FDAT FC81={TOOL_NO 2,BASE_NO 10,IPO_FRAME #BASE,POINT2[] " ",TQ_STATE FALSE}
DECL E6POS XCAux81={X 31.570,Y -15.260,Z 3.110,A 0.010,B 9.930,C -15.040}
DECL E6POS XCDes81={X 32.570,Y -13.780,Z 2.280,A 0.100,B 17.240,C -27.390}
DECL LDAT LCPDATP82={VEL 0.1,ACC 100,APO_DIST 5,APO_FAC 50.0,ORI_TYP #VAR,CIRC_TYP #BASE,JERK_FAC 50.0}
DECL FDAT FP82={TOOL_NO 2,BASE_NO 10,IPO_FRAME #BASE,POINT2[] " ",TQ_STATE FALSE}
DECL E6POS XP82={X 8.690,Y -0.540,Z 2.280,A 0.040,B 12.450,C -29.720}
DECL LDAT LCPDATC83={VEL 0.1,ACC 100,APO_DIST 5,APO_FAC 50.0,ORI_TYP #VAR,CIRC_TYP #BASE,JERK_FAC 50.0}
DECL FDAT FC83={TOOL_NO 2,BASE_NO 10,IPO_FRAME #BASE,POINT2[] " ",TQ_STATE FALSE}
DECL E6POS XCAux83={X -55.000,Y 13.000,Z 2.280,A 0.000,B 0.000,C -32.000}
DECL E6POS XCDes83={X -118.690,Y -0.540,Z 2.280,A -0.040,B -12.450,C -29.720}
DECL LDAT LCPDATC84={VEL 0.5,ACC 100,APO_DIST 5,APO_FAC 50.0,ORI_TYP #VAR,CIRC_TYP #BASE,JERK_FAC 50.0}
DECL FDAT FC84={TOOL_NO 2,BASE_NO 10,IPO_FRAME #BASE,POINT2[] " ",TQ_STATE FALSE}
DECL E6POS XCAux84={X -142.570,Y -13.780,Z 2.280,A -0.100,B -17.240,C -27.390}
DECL E6POS XCDes84={X -142.450,Y -13.950,Z 1.940,A -0.100,B -17.240,C -27.390}
DECL LDAT LCPDATP85={VEL 0.1,ACC 100,APO_DIST 5,APO_FAC 50.0,ORI_TYP #VAR,CIRC_TYP #BASE,JERK_FAC 50.0}
DECL FDAT FP85={TOOL_NO 2,BASE_NO 10,IPO_FRAME #BASE,POINT2[] " ",TQ_STATE FALSE}
DECL E6POS XP85={X -118.610,Y -0.740,Z 1.940,A -0.040,B -12.450,C -29.720}
DECL LDAT LCPDATC86={VEL 0.1,ACC 100,APO_DIST 5,APO_FAC 50.0,ORI_TYP #VAR,CIRC_TYP #BASE,JERK_FAC 50.0}
DECL FDAT FC86={TOOL_NO 2,BASE_NO 10,IPO_FRAME #BASE,POINT2[] " ",TQ_STATE FALSE}
DECL E6POS XCAux86={X -55.000,Y 12.790,Z 1.940,A 0.000,B 0.000,C -32.000}
DECL E6POS XCDes86={X 8.610,Y -0.740,Z 1.940,A 0.040,B 12.450,C -29.720}
DECL LDAT LCPDATC87={VEL 0.5,ACC 100,APO_DIST 5,APO_FAC 50.0,ORI_TYP #VAR,CIRC_TYP #BASE,JERK_FAC 50.0}
DECL FDAT FC87={TOOL_NO 2,BASE_NO 10,IPO_FRAME #BASE,POINT2[] " ",TQ_STATE FALSE}
DECL E6POS XCAux87={X 32.450,Y -13.950,Z 1.940,A 0.100,B 17.240,C -27.390}
DECL E6POS XCDes87={X 31.450,Y -15.430,Z 2.760,A 0.010,B 9.540,C -14.420}
DECL LDAT LCPDATP88={VEL 0.1,ACC 100,APO_DIST 5,APO_FAC 50.0,ORI_TYP #VAR,CIRC_TYP #BASE,JERK_FAC 50.0}
DECL FDAT FP88={TOOL_NO 2,BASE_NO 10,IPO_FRAME #BASE,POINT2[] " ",TQ_STATE FALSE}
DECL E6POS XP88={X 7.880,Y -2.370,Z 2.760,A 0.000,B 6.920,C -15.820}
DECL LDAT LCPDATC89={VEL 0.1,ACC 100,APO_DIST 5,APO_FAC 50.0,ORI_TYP #VAR,CIRC_TYP #BASE,JERK_FAC 50.0}
DECL FDAT FC89={TOOL_NO 2,BASE_NO 10,IPO_FRAME #BASE,POINT2[] " ",TQ_STATE FALSE}
DECL E6POS XCAux89={X -55.000,Y 11.000,Z 2.760,A 0.000,B 0.000,C -17.240}
DECL E6POS XCDes89={X -117.880,Y -2.370,Z 2.760,A -0.000,B -6.920,C -15.820}
DECL LDAT LCPDATC90={VEL 0.5,ACC 100,APO_DIST 5,APO_FAC 50.0,ORI_TYP #VAR,CIRC_TYP #BASE,JERK_FAC 50.0}
DECL FDAT FC90={TOOL_NO 2,BASE_NO 10,IPO_FRAME #BASE,POINT2[] " ",TQ_STATE FALSE}
DECL E6POS XCAux90={X -141.450,Y -15.430,Z 2.760,A -0.010,B -9.540,C -14.420}
DECL E6POS XCDes90={X -140.360,Y -17.040,Z 3.090,A -0.000,B -1.380,C -2.050}
DECL LDAT LCPDATP91={VEL 0.1,ACC 100,APO_DIST 5,APO_FAC 50.0,ORI_TYP #VAR,CIRC_TYP #BASE,JERK_FAC 50.0}
DECL FDAT FP91={TOOL_NO 2,BASE_NO 10,IPO_FRAME #BASE,POINT2[] " ",TQ_STATE FALSE}
DECL E6POS XP91={X -117.090,Y -4.140,Z 3.090,A -0.000,B -1.010,C -2.260}
DECL LDAT LCPDATC92={VEL 0.1,ACC 100,APO_DIST 5,APO_FAC 50.0,ORI_TYP #VAR,CIRC_TYP #BASE,JERK_FAC 50.0}
DECL FDAT FC92={TOOL_NO 2,BASE_NO 10,IPO_FRAME #BASE,POINT2[] " ",TQ_STATE FALSE}
DECL E6POS XCAux92={X -55.000,Y 9.060,Z 3.090,A 0.000,B 0.000,C -2.470}
DECL E6POS XCDes92={X 7.090,Y -4.140,Z 3.090,A 0.000,B 1.010,C -2.260}
DECL LDAT LCPDATC93={VEL 0.5,ACC 100,APO_DIST 5,APO_FAC 50.0,ORI_TYP #VAR,CIRC_TYP #BASE,JERK_FAC 50.0}
DECL FDAT FC93={TOOL_NO 2,BASE_NO 10,IPO_FRAME #BASE,POINT2[] " ",TQ_STATE FALSE}
DECL E6POS XCAux93={X 30.360,Y -17.040,Z 3.090,A 0.000,B 1.380,C -2.050}
DECL E6POS XCDes93={X 30.370,Y -17.040,Z 3.100,A 0.000,B 0.000,C -0.000}
DECL LDAT LCPDATP94={VEL 0.1,ACC 100,APO_DIST 5,APO_FAC 50.0,ORI_TYP #VAR,CIRC_TYP #BASE,JERK_FAC 50.0}
DECL FDAT FP94={TOOL_NO 2,BASE_NO 10,IPO_FRAME #BASE,POINT2[] " ",TQ_STATE FALSE}
DECL E6POS XP94={X 7.090,Y -4.140,Z 3.100,A 0.000,B 0.000,C -0.000}
DECL LDAT LCPDATC95={VEL 0.1,ACC 100,APO_DIST 5,APO_FAC 50.0,ORI_TYP #VAR,CIRC_TYP #BASE,JERK_FAC 50.0}
DECL FDAT FC95={TOOL_NO 2,BASE_NO 10,IPO_FRAME #BASE,POINT2[] " ",TQ_STATE FALSE}
DECL E6POS XCAux95={X -55.000,Y 9.060,Z 3.100,A 0.000,B 0.000,C -0.000}
DECL E6POS XCDes95={X -117.090,Y -4.140,Z 3.100,A 0.000,B 0.000,C -0.000}
DECL LDAT LCPDATC96={VEL 0.5,ACC 100,APO_DIST 5,APO_FAC 50.0,ORI_TYP #VAR,CIRC_TYP #BASE,JERK_FAC 50.0}
DECL FDAT FC96={TOOL_NO 2,BASE_NO 10,IPO_FRAME #BASE,POINT2[] " ",TQ_STATE FALSE}
DECL E6POS XCAux96={X -140.370,Y -17.040,Z 3.100,A 0.000,B 0.000,C -0.000}
DECL E6POS XCDes96={X -139.250,Y -18.700,Z 3.100,A 0.000,B 0.000,C -0.000}
DECL LDAT LCPDATP97={VEL 0.1,ACC 100,APO_DIST 5,APO_FAC 50.0,ORI_TYP #VAR,CIRC_TYP #BASE,JERK_FAC 50.0}
DECL FDAT FP97={TOOL_NO 2,BASE_NO 10,IPO_FRAME #BASE,POINT2[] " ",TQ_STATE FALSE}
DECL E6POS XP97={X -116.280,Y -5.970,Z 3.100,A 0.000,B 0.000,C -0.000}
DECL LDAT LCPDATC98={VEL 0.1,ACC 100,APO_DIST 5,APO_FAC 50.0,ORI_TYP #VAR,CIRC_TYP #BASE,JERK_FAC 50.0}
DECL FDAT FC98={TOOL_NO 2,BASE_NO 10,IPO_FRAME #BASE,POINT2[] " ",TQ_STATE FALSE}
DECL E6POS XCAux98={X -55.000,Y 7.060,Z 3.100,A 0.000,B 0.000,C -0.000}
DECL E6POS XCDes98={X 6.280,Y -5.970,Z 3.100,A 0.000,B 0.000,C -0.000}
DECL LDAT LCPDATC99={VEL 0.5,ACC 100,APO_DIST 5,APO_FAC 50.0,ORI_TYP #VAR,CIRC_TYP #BASE,JERK_FAC 50.0}
DECL FDAT FC99={TOOL_NO 2,BASE_NO 10,IPO_FRAME #BASE,POINT2[] " ",TQ_STATE FALSE}
DECL E6POS XCAux99={X 29.250,Y -18.700,Z 3.100,A 0.000,B 0.000,C -0.000}
DECL E6POS XCDes99={X 28.130,Y -20.360,Z 3.100,A 0.000,B 0.000,C -0.000}
DECL LDAT LCPDATP100={VEL 0.1,ACC 100,APO_DIST 5,APO_FAC 50.0,ORI_TYP #VAR,CIRC_TYP #BASE,JERK_FAC 50.0}
DECL FDAT FP100={TOOL_NO 2,BASE_NO 10,IPO_FRAME #BASE,POINT2[] " ",TQ_STATE FALSE}
DECL E6POS XP100={X 5.470,Y -7.790,Z 3.100,A 0.000,B 0.000,C -0.000}
DECL LDAT LCPDATC101={VEL 0.1,ACC 100,APO_DIST 5,APO_FAC 50.0,ORI_TYP #VAR,CIRC_TYP #BASE,JERK_FAC 50.0}
DECL FDAT FC101={TOOL_NO 2,BASE_NO 10,IPO_FRAME #BASE,POINT2[] " ",TQ_STATE FALSE}
DECL E6POS XCAux101={X -55.000,Y 5.060,Z 3.100,A 0.000,B 0.000,C -0.000}
DECL E6POS XCDes101={X -115.470,Y -7.790,Z 3.100,A 0.000,B 0.000,C -0.000}
DECL LDAT LCPDATC102={VEL 0.5,ACC 100,APO_DIST 5,APO_FAC 50.0,ORI_TYP #VAR,CIRC_TYP #BASE,JERK_FAC 50.0}
DECL FDAT FC102={TOOL_NO 2,BASE_NO 10,IPO_FRAME #BASE,POINT2[] " ",TQ_STATE FALSE}
DECL E6POS XCAux102={X -138.130,Y -20.360,Z 3.100,A 0.000,B 0.000,C -0.000}
DECL E6POS XCDes102={X -137.010,Y -22.010,Z 3.100,A 0.000,B 0.000,C -0.000}
DECL LDAT LCPDATP103={VEL 0.1,ACC 100,APO_DIST 5,APO_FAC 50.0,ORI_TYP #VAR,CIRC_TYP #BASE,JERK_FAC 50.0}
DECL FDAT FP103={TOOL_NO 2,BASE_NO 10,IPO_FRAME #BASE,POINT2[] " ",TQ_STATE FALSE}
DECL E6POS XP103={X -114.650,Y -9.620,Z 3.100,A 0.000,B 0.000,C -0.000}
DECL LDAT LCPDATC104={VEL 0.1,ACC 100,APO_DIST 5,APO_FAC 50.0,ORI_TYP #VAR,CIRC_TYP #BASE,JERK_FAC 50.0}
DECL FDAT FC104={TOOL_NO 2,BASE_NO 10,IPO_FRAME #BASE,POINT2[] " ",TQ_STATE FALSE}
DECL E6POS XCAux104={X -55.000,Y 3.060,Z 3.100,A 0.000,B 0.000,C -0.000}
DECL E6POS XCDes104={X 4.650,Y -9.620,Z 3.100,A 0.000,B 0.000,C -0.000}
DECL LDAT LCPDATC105={VEL 0.5,ACC 100,APO_DIST 5,APO_FAC 50.0,ORI_TYP #VAR,CIRC_TYP #BASE,JERK_FAC 50.0}
DECL FDAT FC105={TOOL_NO 2,BASE_NO 10,IPO_FRAME #BASE,POINT2[] " ",TQ_STATE FALSE}
DECL E6POS XCAux105={X 27.010,Y -22.010,Z 3.100,A 0.000,B 0.000,C -0.000}
DECL E6POS XCDes105={X 25.890,Y -23.670,Z 3.100,A 0.000,B 0.000,C -0.000}
DECL LDAT LCPDATP106={VEL 0.1,ACC 100,APO_DIST 5,APO_FAC 50.0,ORI_TYP #VAR,CIRC_TYP #BASE,JERK_FAC 50.0}
DECL FDAT FP106={TOOL_NO 2,BASE_NO 10,IPO_FRAME #BASE,POINT2[] " ",TQ_STATE FALSE}
DECL E6POS XP106={X 3.840,Y -11.450,Z 3.100,A 0.000,B 0.000,C -0.000}
DECL LDAT LCPDATC107={VEL 0.1,ACC 100,APO_DIST 5,APO_FAC 50.0,ORI_TYP #VAR,CIRC_TYP #BASE,JERK_FAC 50.0}
DECL FDAT FC107={TOOL_NO 2,BASE_NO 10,IPO_FRAME #BASE,POINT2[] " ",TQ_STATE FALSE}
DECL E6POS XCAux107={X -55.000,Y 1.060,Z 3.100,A 0.000,B 0.000,C -0.000}
DECL E6POS XCDes107={X -113.840,Y -11.450,Z 3.100,A 0.000,B 0.000,C -0.000}
DECL LDAT LCPDATC108={VEL 0.5,ACC 100,APO_DIST 5,APO_FAC 50.0,ORI_TYP #VAR,CIRC_TYP #BASE,JERK_FAC 50.0}
DECL FDAT FC108={TOOL_NO 2,BASE_NO 10,IPO_FRAME #BASE,POINT2[] " ",TQ_STATE FALSE}
DECL E6POS XCAux108={X -135.890,Y -23.670,Z 3.100,A 0.000,B 0.000,C -0.000}
DECL E6POS XCDes108={X -134.770,Y -25.330,Z 3.100,A 0.000,B 0.000,C -0.000}
DECL LDAT LCPDATP109={VEL 0.1,ACC 100,APO_DIST 5,APO_FAC 50.0,ORI_TYP #VAR,CIRC_TYP #BASE,JERK_FAC 50.0}
DECL FDAT FP109={TOOL_NO 2,BASE_NO 10,IPO_FRAME #BASE,POINT2[] " ",TQ_STATE FALSE}
DECL E6POS XP109={X -113.020,Y -13.270,Z 3.100,A 0.000,B 0.000,C -0.000}
DECL LDAT LCPDATC110={VEL 0.1,ACC 100,APO_DIST 5,APO_FAC 50.0,ORI_TYP #VAR,CIRC_TYP #BASE,JERK_FAC 50.0}
DECL FDAT FC110={TOOL_NO 2,BASE_NO 10,IPO_FRAME #BASE,POINT2[] " ",TQ_STATE FALSE}
DECL E6POS XCAux110={X -55.000,Y -0.940,Z 3.100,A 0.000,B 0.000,C -0.000}
DECL E6POS XCDes110={X 3.020,Y -13.270,Z 3.100,A 0.000,B 0.000,C -0.000}
DECL LDAT LCPDATC111={VEL 0.5,ACC 100,APO_DIST 5,APO_FAC 50.0,ORI_TYP #VAR,CIRC_TYP #BASE,JERK_FAC 50.0}
DECL FDAT FC111={TOOL_NO 2,BASE_NO 10,IPO_FRAME #BASE,POINT2[] " ",TQ_STATE FALSE}
DECL E6POS XCAux111={X 24.770,Y -25.330,Z 3.100,A 0.000,B 0.000,C -0.000}
DECL E6POS XCDes111={X 23.660,Y -26.990,Z 3.100,A 0.000,B 0.000,C -0.000}
DECL LDAT LCPDATP112={VEL 0.1,ACC 100,APO_DIST 5,APO_FAC 50.0,ORI_TYP #VAR,CIRC_TYP #BASE,JERK_FAC 50.0}
DECL FDAT FP112={TOOL_NO 2,BASE_NO 10,IPO_FRAME #BASE,POINT2[] " ",TQ_STATE FALSE}
DECL E6POS XP112={X 2.210,Y -15.100,Z 3.100,A 0.000,B 0.000,C -0.000}
DECL LDAT LCPDATC113={VEL 0.1,ACC 100,APO_DIST 5,APO_FAC 50.0,ORI_TYP #VAR,CIRC_TYP #BASE,JERK_FAC 50.0}
DECL FDAT FC113={TOOL_NO 2,BASE_NO 10,IPO_FRAME #BASE,POINT2[] " ",TQ_STATE FALSE}
DECL E6POS XCAux113={X -55.000,Y -2.940,Z 3.100,A 0.000,B 0.000,C -0.000}
DECL E6POS XCDes113={X -112.210,Y -15.100,Z 3.100,A 0.000,B 0.000,C -0.000}
DECL LDAT LCPDATC114={VEL 0.5,ACC 100,APO_DIST 5,APO_FAC 50.0,ORI_TYP #VAR,CIRC_TYP #BASE,JERK_FAC 50.0}
DECL FDAT FC114={TOOL_NO 2,BASE_NO 10,IPO_FRAME #BASE,POINT2[] " ",TQ_STATE FALSE}
DECL E6POS XCAux114={X -133.660,Y -26.990,Z 3.100,A 0.000,B 0.000,C -0.000}
DECL E6POS XCDes114={X -132.540,Y -28.650,Z 3.100,A 0.000,B 0.000,C -0.000}
DECL LDAT LCPDATP115={VEL 0.1,ACC 100,APO_DIST 5,APO_FAC 50.0,ORI_TYP #VAR,CIRC_TYP #BASE,JERK_FAC 50.0}
DECL FDAT FP115={TOOL_NO 2,BASE_NO 10,IPO_FRAME #BASE,POINT2[] " ",TQ_STATE FALSE}
DECL E6POS XP115={X -111.400,Y -16.930,Z 3.100,A 0.000,B 0.000,C -0.000}
DECL LDAT LCPDATC116={VEL 0.1,ACC 100,APO_DIST 5,APO_FAC 50.0,ORI_TYP #VAR,CIRC_TYP #BASE,JERK_FAC 50.0}
DECL FDAT FC116={TOOL_NO 2,BASE_NO 10,IPO_FRAME #BASE,POINT2[] " ",TQ_STATE FALSE}
DECL E6POS XCAux116={X -55.000,Y -4.940,Z 3.100,A 0.000,B 0.000,C -0.000}
DECL E6POS XCDes116={X 1.400,Y -16.930,Z 3.100,A 0.000,B 0.000,C -0.000}
DECL LDAT LCPDATC117={VEL 0.5,ACC 100,APO_DIST 5,APO_FAC 50.0,ORI_TYP #VAR,CIRC_TYP #BASE,JERK_FAC 50.0}
DECL FDAT FC117={TOOL_NO 2,BASE_NO 10,IPO_FRAME #BASE,POINT2[] " ",TQ_STATE FALSE}
DECL E6POS XCAux117={X 22.540,Y -28.650,Z 3.100,A 0.000,B 0.000,C -0.000}
DECL E6POS XCDes117={X 22.000,Y -29.450,Z 3.100,A 0.000,B 0.070,C -0.110}
DECL LDAT LCPDATP118={VEL 0.1,ACC 100,APO_DIST 5,APO_FAC 50.0,ORI_TYP #VAR,CIRC_TYP #BASE,JERK_FAC 50.0}
DECL FDAT FP118={TOOL_NO 2,BASE_NO 10,IPO_FRAME #BASE,POINT2[] " ",TQ_STATE FALSE}
DECL E6POS XP118={X 1.000,Y -17.810,Z 3.100,A 0.000,B 0.050,C -0.120}
DECL LDAT LCPDATC119={VEL 0.1,ACC 100,APO_DIST 5,APO_FAC 50.0,ORI_TYP #VAR,CIRC_TYP #BASE,JERK_FAC 50.0}
DECL FDAT FC119={TOOL_NO 2,BASE_NO 10,IPO_FRAME #BASE,POINT2[] " ",TQ_STATE FALSE}
DECL E6POS XCAux119={X -55.000,Y -5.910,Z 3.100,A 0.000,B 0.000,C -0.130}
DECL E6POS XCDes119={X -111.000,Y -17.810,Z 3.100,A -0.000,B -0.050,C -0.120}
DECL LDAT LCPDATC120={VEL 0.5,ACC 100,APO_DIST 5,APO_FAC 50.0,ORI_TYP #VAR,CIRC_TYP #BASE,JERK_FAC 50.0}
DECL FDAT FC120={TOOL_NO 2,BASE_NO 10,IPO_FRAME #BASE,POINT2[] " ",TQ_STATE FALSE}
DECL E6POS XCAux120={X -132.000,Y -29.450,Z 3.100,A -0.000,B -0.070,C -0.110}
DECL E6POS XCDes120={X -130.900,Y -31.070,Z 2.850,A -0.000,B 8.120,C 12.220}
DECL LDAT LCPDATP121={VEL 0.1,ACC 100,APO_DIST 5,APO_FAC 50.0,ORI_TYP #VAR,CIRC_TYP #BASE,JERK_FAC 50.0}
DECL FDAT FP121={TOOL_NO 2,BASE_NO 10,IPO_FRAME #BASE,POINT2[] " ",TQ_STATE FALSE}
DECL E6POS XP121={X -110.210,Y -19.600,Z 2.850,A -0.000,B 5.900,C 13.420}
DECL LDAT LCPDATC122={VEL 0.1,ACC 100,APO_DIST 5,APO_FAC 50.0,ORI_TYP #VAR,CIRC_TYP #BASE,JERK_FAC 50.0}
DECL FDAT FC122={TOOL_NO 2,BASE_NO 10,IPO_FRAME #BASE,POINT2[] " ",TQ_STATE FALSE}
DECL E6POS XCAux122={X -55.000,Y -7.860,Z 2.850,A 0.000,B 0.000,C 14.640}
DECL E6POS XCDes122={X 0.210,Y -19.600,Z 2.850,A 0.000,B -5.900,C 13.420}
DECL LDAT LCPDATC123={VEL 0.5,ACC 100,APO_DIST 5,APO_FAC 50.0,ORI_TYP #VAR,CIRC_TYP #BASE,JERK_FAC 50.0}
DECL FDAT FC123={TOOL_NO 2,BASE_NO 10,IPO_FRAME #BASE,POINT2[] " ",TQ_STATE FALSE}
DECL E6POS XCAux123={X 20.900,Y -31.070,Z 2.850,A 0.000,B -8.120,C 12.220}
DECL E6POS XCDes123={X 19.880,Y -32.580,Z 2.110,A 0.070,B -15.930,C 25.040}
DECL LDAT LCPDATP124={VEL 0.1,ACC 100,APO_DIST 5,APO_FAC 50.0,ORI_TYP #VAR,CIRC_TYP #BASE,JERK_FAC 50.0}
DECL FDAT FP124={TOOL_NO 2,BASE_NO 10,IPO_FRAME #BASE,POINT2[] " ",TQ_STATE FALSE}
DECL E6POS XP124={X -0.530,Y -21.260,Z 2.110,A 0.030,B -11.520,C 27.240}
DECL LDAT LCPDATC125={VEL 0.1,ACC 100,APO_DIST 5,APO_FAC 50.0,ORI_TYP #VAR,CIRC_TYP #BASE,JERK_FAC 50.0}
DECL FDAT FC125={TOOL_NO 2,BASE_NO 10,IPO_FRAME #BASE,POINT2[] " ",TQ_STATE FALSE}
DECL E6POS XCAux125={X -55.000,Y -9.690,Z 2.110,A 0.000,B 0.000,C 29.400}
DECL E6POS XCDes125={X -109.470,Y -21.260,Z 2.110,A -0.030,B 11.520,C 27.240}
DECL LDAT LCPDATC126={VEL 0.5,ACC 100,APO_DIST 5,APO_FAC 50.0,ORI_TYP #VAR,CIRC_TYP #BASE,JERK_FAC 50.0}
DECL FDAT FC126={TOOL_NO 2,BASE_NO 10,IPO_FRAME #BASE,POINT2[] " ",TQ_STATE FALSE}
DECL E6POS XCAux126={X -129.880,Y -32.580,Z 2.110,A -0.070,B 15.930,C 25.040}
DECL E6POS XCDes126={X -129.890,Y -32.570,Z 1.660,A -0.090,B 16.750,C 26.510}
DECL LDAT LCPDATP127={VEL 0.1,ACC 100,APO_DIST 5,APO_FAC 50.0,ORI_TYP #VAR,CIRC_TYP #BASE,JERK_FAC 50.0}
DECL FDAT FP127={TOOL_NO 2,BASE_NO 10,IPO_FRAME #BASE,POINT2[] " ",TQ_STATE FALSE}
DECL E6POS XP127={X -109.480,Y -21.250,Z 1.660,A -0.040,B 12.100,C 28.790}
DECL LDAT LCPDATC128={VEL 0.1,ACC 100,APO_DIST 5,APO_FAC 50.0,ORI_TYP #VAR,CIRC_TYP #BASE,JERK_FAC 50.0}
DECL FDAT FC128={TOOL_NO 2,BASE_NO 10,IPO_FRAME #BASE,POINT2[] " ",TQ_STATE FALSE}
DECL E6POS XCAux128={X -55.000,Y -9.670,Z 1.660,A 0.000,B 0.000,C 31.030}
DECL E6POS XCDes128={X -0.520,Y -21.250,Z 1.660,A 0.040,B -12.100,C 28.790}
DECL LDAT LCPDATC129={VEL 0.5,ACC 100,APO_DIST 5,APO_FAC 50.0,ORI_TYP #VAR,CIRC_TYP #BASE,JERK_FAC 50.0}
DECL FDAT FC129={TOOL_NO 2,BASE_NO 10,IPO_FRAME #BASE,POINT2[] " ",TQ_STATE FALSE}
DECL E6POS XCAux129={X 19.890,Y -32.570,Z 1.660,A 0.090,B -16.750,C 26.510}
DECL E6POS XCDes129={X 20.900,Y -31.070,Z 2.440,A 0.010,B -8.570,C 12.920}
DECL LDAT LCPDATP130={VEL 0.1,ACC 100,APO_DIST 5,APO_FAC 50.0,ORI_TYP #VAR,CIRC_TYP #BASE,JERK_FAC 50.0}
DECL FDAT FP130={TOOL_NO 2,BASE_NO 10,IPO_FRAME #BASE,POINT2[] " ",TQ_STATE FALSE}
DECL E6POS XP130={X 0.210,Y -19.600,Z 2.440,A 0.000,B -6.230,C 14.180}
DECL LDAT LCPDATC131={VEL 0.1,ACC 100,APO_DIST 5,APO_FAC 50.0,ORI_TYP #VAR,CIRC_TYP #BASE,JERK_FAC 50.0}
DECL FDAT FC131={TOOL_NO 2,BASE_NO 10,IPO_FRAME #BASE,POINT2[] " ",TQ_STATE FALSE}
DECL E6POS XCAux131={X -55.000,Y -7.860,Z 2.440,A 0.000,B 0.000,C 15.460}
DECL E6POS XCDes131={X -110.210,Y -19.600,Z 2.440,A -0.000,B 6.230,C 14.180}
DECL LDAT LCPDATC132={VEL 0.5,ACC 100,APO_DIST 5,APO_FAC 50.0,ORI_TYP #VAR,CIRC_TYP #BASE,JERK_FAC 50.0}
DECL FDAT FC132={TOOL_NO 2,BASE_NO 10,IPO_FRAME #BASE,POINT2[] " ",TQ_STATE FALSE}
DECL E6POS XCAux132={X -130.900,Y -31.070,Z 2.440,A -0.010,B 8.570,C 12.920}
DECL E6POS XCDes132={X -131.990,Y -29.450,Z 2.700,A -0.000,B -0.060,C -0.090}
DECL LDAT LCPDATP133={VEL 0.1,ACC 100,APO_DIST 5,APO_FAC 50.0,ORI_TYP #VAR,CIRC_TYP #BASE,JERK_FAC 50.0}
DECL FDAT FP133={TOOL_NO 2,BASE_NO 10,IPO_FRAME #BASE,POINT2[] " ",TQ_STATE FALSE}
DECL E6POS XP133={X -111.000,Y -17.820,Z 2.700,A -0.000,B -0.040,C -0.090}
DECL LDAT LCPDATC134={VEL 0.1,ACC 100,APO_DIST 5,APO_FAC 50.0,ORI_TYP #VAR,CIRC_TYP #BASE,JERK_FAC 50.0}
DECL FDAT FC134={TOOL_NO 2,BASE_NO 10,IPO_FRAME #BASE,POINT2[] " ",TQ_STATE FALSE}
DECL E6POS XCAux134={X -55.000,Y -5.910,Z 2.700,A 0.000,B 0.000,C -0.100}
DECL E6POS XCDes134={X 1.000,Y -17.820,Z 2.700,A 0.000,B 0.040,C -0.090}
DECL LDAT LCPDATC135={VEL 0.5,ACC 100,APO_DIST 5,APO_FAC 50.0,ORI_TYP #VAR,CIRC_TYP #BASE,JERK_FAC 50.0}
DECL FDAT FC135={TOOL_NO 2,BASE_NO 10,IPO_FRAME #BASE,POINT2[] " ",TQ_STATE FALSE}
DECL E6POS XCAux135={X 21.990,Y -29.450,Z 2.700,A 0.000,B 0.060,C -0.090}
DECL E6POS XCDes135={X 22.410,Y -28.830,Z 2.700,A 0.000,B 0.000,C -0.000}
DECL LDAT LCPDATP136={VEL 0.1,ACC 100,APO_DIST 5,APO_FAC 50.0,ORI_TYP #VAR,CIRC_TYP #BASE,JERK_FAC 50.0}
DECL FDAT FP136={TOOL_NO 2,BASE_NO 10,IPO_FRAME #BASE,POINT2[] " ",TQ_STATE FALSE}
DECL E6POS XP136={X 1.310,Y -17.130,Z 2.700,A 0.000,B 0.000,C -0.000}
DECL LDAT LCPDATC137={VEL 0.1,ACC 100,APO_DIST 5,APO_FAC 50.0,ORI_TYP #VAR,CIRC_TYP #BASE,JERK_FAC 50.0}
DECL FDAT FC137={TOOL_NO 2,BASE_NO 10,IPO_FRAME #BASE,POINT2[] " ",TQ_STATE FALSE}
DECL E6POS XCAux137={X -55.000,Y -5.160,Z 2.700,A 0.000,B 0.000,C -0.000}
DECL E6POS XCDes137={X -111.310,Y -17.130,Z 2.700,A 0.000,B 0.000,C -0.000}
DECL LDAT LCPDATC138={VEL 0.5,ACC 100,APO_DIST 5,APO_FAC 50.0,ORI_TYP #VAR,CIRC_TYP #BASE,JERK_FAC 50.0}
DECL FDAT FC138={TOOL_NO 2,BASE_NO 10,IPO_FRAME #BASE,POINT2[] " ",TQ_STATE FALSE}
DECL E6POS XCAux138={X -132.410,Y -28.830,Z 2.700,A 0.000,B 0.000,C -0.000}
DECL E6POS XCDes138={X -133.530,Y -27.170,Z 2.700,A 0.000,B 0.000,C -0.000}
DECL LDAT LCPDATP139={VEL 0.1,ACC 100,APO_DIST 5,APO_FAC 50.0,ORI_TYP #VAR,CIRC_TYP #BASE,JERK_FAC 50.0}
DECL FDAT FP139={TOOL_NO 2,BASE_NO 10,IPO_FRAME #BASE,POINT2[] " ",TQ_STATE FALSE}
DECL E6POS XP139={X -112.120,Y -15.300,Z 2.700,A 0.000,B 0.000,C -0.000}
DECL LDAT LCPDATC140={VEL 0.1,ACC 100,APO_DIST 5,APO_FAC 50.0,ORI_TYP #VAR,CIRC_TYP #BASE,JERK_FAC 50.0}
DECL FDAT FC140={TOOL_NO 2,BASE_NO 10,IPO_FRAME #BASE,POINT2[] " ",TQ_STATE FALSE}
DECL E6POS XCAux140={X -55.000,Y -3.160,Z 2.700,A 0.000,B 0.000,C -0.000}
DECL E6POS XCDes140={X 2.120,Y -15.300,Z 2.700,A 0.000,B 0.000,C -0.000}
DECL LDAT LCPDATC141={VEL 0.5,ACC 100,APO_DIST 5,APO_FAC 50.0,ORI_TYP #VAR,CIRC_TYP #BASE,JERK_FAC 50.0}
DECL FDAT FC141={TOOL_NO 2,BASE_NO 10,IPO_FRAME #BASE,POINT2[] " ",TQ_STATE FALSE}
DECL E6POS XCAux141={X 23.530,Y -27.170,Z 2.700,A 0.000,B 0.000,C -0.000}
DECL E6POS XCDes141={X 24.650,Y -25.510,Z 2.700,A 0.000,B 0.000,C -0.000}
DECL LDAT LCPDATP142={VEL 0.1,ACC 100,APO_DIST 5,APO_FAC 50.0,ORI_TYP #VAR,CIRC_TYP #BASE,JERK_FAC 50.0}
DECL FDAT FP142={TOOL_NO 2,BASE_NO 10,IPO_FRAME #BASE,POINT2[] " ",TQ_STATE FALSE}
DECL E6POS XP142={X 2.930,Y -13.480,Z 2.700,A 0.000,B 0.000,C -0.000}
DECL LDAT LCPDATC143={VEL 0.1,ACC 100,APO_DIST 5,APO_FAC 50.0,ORI_TYP #VAR,CIRC_TYP #BASE,JERK_FAC 50.0}
DECL FDAT FC143={TOOL_NO 2,BASE_NO 10,IPO_FRAME #BASE,POINT2[] " ",TQ_STATE FALSE}
DECL E6POS XCAux143={X -55.000,Y -1.160,Z 2.700,A 0.000,B 0.000,C -0.000}
DECL E6POS XCDes143={X -112.930,Y -13.480,Z 2.700,A 0.000,B 0.000,C -0.000}
DECL LDAT LCPDATC144={VEL 0.5,ACC 100,APO_DIST 5,APO_FAC 50.0,ORI_TYP #VAR,CIRC_TYP #BASE,JERK_FAC 50.0}
DECL FDAT FC144={TOOL_NO 2,BASE_NO 10,IPO_FRAME #BASE,POINT2[] " ",TQ_STATE FALSE}
DECL E6POS XCAux144={X -134.650,Y -25.510,Z 2.700,A 0.000,B 0.000,C -0.000}
DECL E6POS XCDes144={X -135.770,Y -23.860,Z 2.700,A 0.000,B 0.000,C -0.000}
DECL LDAT LCPDATP145={VEL 0.1,ACC 100,APO_DIST 5,APO_FAC 50.0,ORI_TYP #VAR,CIRC_TYP #BASE,JERK_FAC 50.0}
DECL FDAT FP145={TOOL_NO 2,BASE_NO 10,IPO_FRAME #BASE,POINT2[] " ",TQ_STATE FALSE}
DECL E6POS XP145={X -113.750,Y -11.650,Z 2.700,A 0.000,B 0.000,C -0.000}
DECL LDAT LCPDATC146={VEL 0.1,ACC 100,APO_DIST 5,APO_FAC 50.0,ORI_TYP #VAR,CIRC_TYP #BASE,JERK_FAC 50.0}
DECL FDAT FC146={TOOL_NO 2,BASE_NO 10,IPO_FRAME #BASE,POINT2[] " ",TQ_STATE FALSE}
DECL E6POS XCAux146={X -55.000,Y 0.840,Z 2.700,A 0.000,B 0.000,C -0.000}
DECL E6POS XCDes146={X 3.750,Y -11.650,Z 2.700,A 0.000,B 0.000,C -0.000}
DECL LDAT LCPDATC147={VEL 0.5,ACC 100,APO_DIST 5,APO_FAC 50.0,ORI_TYP #VAR,CIRC_TYP #BASE,JERK_FAC 50.0}
DECL FDAT FC147={TOOL_NO 2,BASE_NO 10,IPO_FRAME #BASE,POINT2[] " ",TQ_STATE FALSE}
DECL E6POS XCAux147={X 25.770,Y -23.860,Z 2.700,A 0.000,B 0.000,C -0.000}
DECL E6POS XCDes147={X 26.890,Y -22.200,Z 2.700,A 0.000,B 0.000,C -0.000}
DECL LDAT LCPDATP148={VEL 0.1,ACC 100,APO_DIST 5,APO_FAC 50.0,ORI_TYP #VAR,CIRC_TYP #BASE,JERK_FAC 50.0}
DECL FDAT FP148={TOOL_NO 2,BASE_NO 10,IPO_FRAME #BASE,POINT2[] " ",TQ_STATE FALSE}
DECL E6POS XP148={X 4.560,Y -9.820,Z 2.700,A 0.000,B 0.000,C -0.000}
DECL LDAT LCPDATC149={VEL 0.1,ACC 100,APO_DIST 5,APO_FAC 50.0,ORI_TYP #VAR,CIRC_TYP #BASE,JERK_FAC 50.0}
DECL FDAT FC149={TOOL_NO 2,BASE_NO 10,IPO_FRAME #BASE,POINT2[] " ",TQ_STATE FALSE}
DECL E6POS XCAux149={X -55.000,Y 2.840,Z 2.700,A 0.000,B 0.000,C -0.000}
DECL E6POS XCDes149={X -114.560,Y -9.820,Z 2.700,A 0.000,B 0.000,C -0.000}
DECL LDAT LCPDATC150={VEL 0.5,ACC 100,APO_DIST 5,APO_FAC 50.0,ORI_TYP #VAR,CIRC_TYP #BASE,JERK_FAC 50.0}
DECL FDAT FC150={TOOL_NO 2,BASE_NO 10,IPO_FRAME #BASE,POINT2[] " ",TQ_STATE FALSE}
DECL E6POS XCAux150={X -136.890,Y -22.200,Z 2.700,A 0.000,B 0.000,C -0.000}
DECL E6POS XCDes150={X -138.000,Y -20.540,Z 2.700,A 0.000,B 0.000,C -0.000}
DECL LDAT LCPDATP151={VEL 0.1,ACC 100,APO_DIST 5,APO_FAC 50.0,ORI_TYP #VAR,CIRC_TYP #BASE,JERK_FAC 50.0}
DECL FDAT FP151={TOOL_NO 2,BASE_NO 10,IPO_FRAME #BASE,POINT2[] " ",TQ_STATE FALSE}
DECL E6POS XP151={X -115.370,Y -8.000,Z 2.700,A 0.000,B 0.000,C -0.000}
DECL LDAT LCPDATC152={VEL 0.1,ACC 100,APO_DIST 5,APO_FAC 50.0,ORI_TYP #VAR,CIRC_TYP #BASE,JERK_FAC 50.0}
DECL FDAT FC152={TOOL_NO 2,BASE_NO 10,IPO_FRAME #BASE,POINT2[] " ",TQ_STATE FALSE}
DECL E6POS XCAux152={X -55.000,Y 4.840,Z 2.700,A 0.000,B 0.000,C -0.000}
DECL E6POS XCDes152={X 5.370,Y -8.000,Z 2.700,A 0.000,B 0.000,C -0.000}
DECL LDAT LCPDATC153={VEL 0.5,ACC 100,APO_DIST 5,APO_FAC 50.0,ORI_TYP #VAR,CIRC_TYP #BASE,JERK_FAC 50.0}
DECL FDAT FC153={TOOL_NO 2,BASE_NO 10,IPO_FRAME #BASE,POINT2[] " ",TQ_STATE FALSE}
DECL E6POS XCAux153={X 28.000,Y -20.540,Z 2.700,A 0.000,B 0.000,C -0.000}
DECL E6POS XCDes153={X 29.120,Y -18.880,Z 2.700,A 0.000,B 0.000,C -0.000}
DECL LDAT LCPDATP154={VEL 0.1,ACC 100,APO_DIST 5,APO_FAC 50.0,ORI_TYP #VAR,CIRC_TYP #BASE,JERK_FAC 50.0}
DECL FDAT FP154={TOOL_NO 2,BASE_NO 10,IPO_FRAME #BASE,POINT2[] " ",TQ_STATE FALSE}
DECL E6POS XP154={X 6.190,Y -6.170,Z 2.700,A 0.000,B 0.000,C -0.000}
DECL LDAT LCPDATC155={VEL 0.1,ACC 100,APO_DIST 5,APO_FAC 50.0,ORI_TYP #VAR,CIRC_TYP #BASE,JERK_FAC 50.0}
DECL FDAT FC155={TOOL_NO 2,BASE_NO 10,IPO_FRAME #BASE,POINT2[] " ",TQ_STATE FALSE}
DECL E6POS XCAux155={X -55.000,Y 6.840,Z 2.700,A 0.000,B 0.000,C -0.000}
DECL E6POS XCDes155={X -116.190,Y -6.170,Z 2.700,A 0.000,B 0.000,C -0.000}
DECL LDAT LCPDATC156={VEL 0.5,ACC 100,APO_DIST 5,APO_FAC 50.0,ORI_TYP #VAR,CIRC_TYP #BASE,JERK_FAC 50.0}
DECL FDAT FC156={TOOL_NO 2,BASE_NO 10,IPO_FRAME #BASE,POINT2[] " ",TQ_STATE FALSE}
DECL E6POS XCAux156={X -139.120,Y -18.880,Z 2.700,A 0.000,B 0.000,C -0.000}
DECL E6POS XCDes156={X -140.240,Y -17.220,Z 2.700,A 0.000,B 0.000,C -0.000}
DECL LDAT LCPDATP157={VEL 0.1,ACC 100,APO_DIST 5,APO_FAC 50.0,ORI_TYP #VAR,CIRC_TYP #BASE,JERK_FAC 50.0}
DECL FDAT FP157={TOOL_NO 2,BASE_NO 10,IPO_FRAME #BASE,POINT2[] " ",TQ_STATE FALSE}
DECL E6POS XP157={X -117.000,Y -4.340,Z 2.700,A 0.000,B 0.000,C -0.000}
DECL LDAT LCPDATC158={VEL 0.1,ACC 100,APO_DIST 5,APO_FAC 50.0,ORI_TYP #VAR,CIRC_TYP #BASE,JERK_FAC 50.0}
DECL FDAT FC158={TOOL_NO 2,BASE_NO 10,IPO_FRAME #BASE,POINT2[] " ",TQ_STATE FALSE}
DECL E6POS XCAux158={X -55.000,Y 8.840,Z 2.700,A 0.000,B 0.000,C -0.000}
DECL E6POS XCDes158={X 7.000,Y -4.340,Z 2.700,A 0.000,B 0.000,C -0.000}
DECL LDAT LCPDATC159={VEL 0.5,ACC 100,APO_DIST 5,APO_FAC 50.0,ORI_TYP #VAR,CIRC_TYP #BASE,JERK_FAC 50.0}
DECL FDAT FC159={TOOL_NO 2,BASE_NO 10,IPO_FRAME #BASE,POINT2[] " ",TQ_STATE FALSE}
DECL E6POS XCAux159={X 30.240,Y -17.220,Z 2.700,A 0.000,B 0.000,C -0.000}
DECL E6POS XCDes159={X 30.240,Y -17.230,Z 2.700,A 0.000,B 0.490,C -0.720}
DECL LDAT LCPDATP160={VEL 0.1,ACC 100,APO_DIST 5,APO_FAC 50.0,ORI_TYP #VAR,CIRC_TYP #BASE,JERK_FAC 50.0}
DECL FDAT FP160={TOOL_NO 2,BASE_NO 10,IPO_FRAME #BASE,POINT2[] " ",TQ_STATE FALSE}
DECL E6POS XP160={X 7.000,Y -4.340,Z 2.700,A 0.000,B 0.350,C -0.790}
DECL LDAT LCPDATC161={VEL 0.1,ACC 100,APO_DIST 5,APO_FAC 50.0,ORI_TYP #VAR,CIRC_TYP #BASE,JERK_FAC 50.0}
DECL FDAT FC161={TOOL_NO 2,BASE_NO 10,IPO_FRAME #BASE,POINT2[] " ",TQ_STATE FALSE}
DECL E6POS XCAux161={X -55.000,Y 8.830,Z 2.700,A 0.000,B 0.000,C -0.870}
DECL E6POS XCDes161={X -117.000,Y -4.340,Z 2.700,A -0.000,B -0.350,C -0.790}
DECL LDAT LCPDATC162={VEL 0.5,ACC 100,APO_DIST 5,APO_FAC 50.0,ORI_TYP #VAR,CIRC_TYP #BASE,JERK_FAC 50.0}
DECL FDAT FC162={TOOL_NO 2,BASE_NO 10,IPO_FRAME #BASE,POINT2[] " ",TQ_STATE FALSE}
DECL E6POS XCAux162={X -140.240,Y -17.230,Z 2.700,A -0.000,B -0.490,C -0.720}
DECL E6POS XCDes162={X -141.330,Y -15.610,Z 2.400,A -0.010,B -9.100,C -13.740}
DECL LDAT LCPDATP163={VEL 0.1,ACC 100,APO_DIST 5,APO_FAC 50.0,ORI_TYP #VAR,CIRC_TYP #BASE,JERK_FAC 50.0}
DECL FDAT FP163={TOOL_NO 2,BASE_NO 10,IPO_FRAME #BASE,POINT2[] " ",TQ_STATE FALSE}
DECL E6POS XP163={X -117.790,Y -2.570,Z 2.400,A -0.000,B -6.610,C -15.080}
DECL LDAT LCPDATC164={VEL 0.1,ACC 100,APO_DIST 5,APO_FAC 50.0,ORI_TYP #VAR,CIRC_TYP #BASE,JERK_FAC 50.0}
DECL FDAT FC164={TOOL_NO 2,BASE_NO 10,IPO_FRAME #BASE,POINT2[] " ",TQ_STATE FALSE}
DECL E6POS XCAux164={X -55.000,Y 10.780,Z 2.400,A 0.000,B 0.000,C -16.430}
DECL E6POS XCDes164={X 7.790,Y -2.570,Z 2.400,A 0.000,B 6.610,C -15.080}
DECL LDAT LCPDATC165={VEL 0.5,ACC 100,APO_DIST 5,APO_FAC 50.0,ORI_TYP #VAR,CIRC_TYP #BASE,JERK_FAC 50.0}
DECL FDAT FC165={TOOL_NO 2,BASE_NO 10,IPO_FRAME #BASE,POINT2[] " ",TQ_STATE FALSE}
DECL E6POS XCAux165={X 31.330,Y -15.610,Z 2.400,A 0.010,B 9.100,C -13.740}
DECL E6POS XCDes165={X 32.330,Y -14.130,Z 1.600,A 0.100,B 17.240,C -27.390}
DECL LDAT LCPDATP166={VEL 0.1,ACC 100,APO_DIST 5,APO_FAC 50.0,ORI_TYP #VAR,CIRC_TYP #BASE,JERK_FAC 50.0}
DECL FDAT FP166={TOOL_NO 2,BASE_NO 10,IPO_FRAME #BASE,POINT2[] " ",TQ_STATE FALSE}
DECL E6POS XP166={X 8.520,Y -0.930,Z 1.600,A 0.040,B 12.450,C -29.720}
DECL LDAT LCPDATC167={VEL 0.1,ACC 100,APO_DIST 5,APO_FAC 50.0,ORI_TYP #VAR,CIRC_TYP #BASE,JERK_FAC 50.0}
DECL FDAT FC167={TOOL_NO 2,BASE_NO 10,IPO_FRAME #BASE,POINT2[] " ",TQ_STATE FALSE}
DECL E6POS XCAux167={X -55.000,Y 12.570,Z 1.600,A 0.000,B 0.000,C -32.000}
DECL E6POS XCDes167={X -118.520,Y -0.930,Z 1.600,A -0.040,B -12.450,C -29.720}
DECL LDAT LCPDATC168={VEL 0.5,ACC 100,APO_DIST 5,APO_FAC 50.0,ORI_TYP #VAR,CIRC_TYP #BASE,JERK_FAC 50.0}
DECL FDAT FC168={TOOL_NO 2,BASE_NO 10,IPO_FRAME #BASE,POINT2[] " ",TQ_STATE FALSE}
DECL E6POS XCAux168={X -142.330,Y -14.130,Z 1.600,A -0.100,B -17.240,C -27.390}
DECL E6POS XCDes168={X -141.210,Y -15.790,Z 2.050,A -0.010,B -8.620,C -12.980}
DECL LDAT LCPDATP169={VEL 0.1,ACC 100,APO_DIST 5,APO_FAC 50.0,ORI_TYP #VAR,CIRC_TYP #BASE,JERK_FAC 50.0}
DECL FDAT FP169={TOOL_NO 2,BASE_NO 10,IPO_FRAME #BASE,POINT2[] " ",TQ_STATE FALSE}
DECL E6POS XP169={X -117.700,Y -2.760,Z 2.050,A -0.000,B -6.260,C -14.250}
DECL LDAT LCPDATC170={VEL 0.1,ACC 100,APO_DIST 5,APO_FAC 50.0,ORI_TYP #VAR,CIRC_TYP #BASE,JERK_FAC 50.0}
DECL FDAT FC170={TOOL_NO 2,BASE_NO 10,IPO_FRAME #BASE,POINT2[] " ",TQ_STATE FALSE}
DECL E6POS XCAux170={X -55.000,Y 10.560,Z 2.050,A 0.000,B 0.000,C -15.540}
DECL E6POS XCDes170={X 7.700,Y -2.760,Z 2.050,A 0.000,B 6.260,C -14.250}
DECL LDAT LCPDATC171={VEL 0.5,ACC 100,APO_DIST 5,APO_FAC 50.0,ORI_TYP #VAR,CIRC_TYP #BASE,JERK_FAC 50.0}
DECL FDAT FC171={TOOL_NO 2,BASE_NO 10,IPO_FRAME #BASE,POINT2[] " ",TQ_STATE FALSE}
DECL E6POS XCAux171={X 31.210,Y -15.790,Z 2.050,A 0.010,B 8.620,C -12.980}
DECL E6POS XCDes171={X 31.220,Y -15.770,Z 2.300,A 0.000,B 0.000,C -0.000}
DECL LDAT LCPDATP172={VEL 0.1,ACC 100,APO_DIST 5,APO_FAC 50.0,ORI_TYP #VAR,CIRC_TYP #BASE,JERK_FAC 50.0}
DECL FDAT FP172={TOOL_NO 2,BASE_NO 10,IPO_FRAME #BASE,POINT2[] " ",TQ_STATE FALSE}
DECL E6POS XP172={X 7.710,Y -2.740,Z 2.300,A 0.000,B 0.000,C -0.000}
DECL LDAT LCPDATC173={VEL 0.1,ACC 100,APO_DIST 5,APO_FAC 50.0,ORI_TYP #VAR,CIRC_TYP #BASE,JERK_FAC 50.0}
DECL FDAT FC173={TOOL_NO 2,BASE_NO 10,IPO_FRAME #BASE,POINT2[] " ",TQ_STATE FALSE}
DECL E6POS XCAux173={X -55.000,Y 10.590,Z 2.300,A 0.000,B 0.000,C -0.000}
DECL E6POS XCDes173={X -117.710,Y -2.740,Z 2.300,A 0.000,B 0.000,C -0.000}
DECL LDAT LCPDATC174={VEL 0.5,ACC 100,APO_DIST 5,APO_FAC 50.0,ORI_TYP #VAR,CIRC_TYP #BASE,JERK_FAC 50.0}
DECL FDAT FC174={TOOL_NO 2,BASE_NO 10,IPO_FRAME #BASE,POINT2[] " ",TQ_STATE FALSE}
DECL E6POS XCAux174={X -141.220,Y -15.770,Z 2.300,A 0.000,B 0.000,C -0.000}
DECL E6POS XCDes174={X -140.100,Y -17.430,Z 2.300,A 0.000,B 0.000,C -0.000}
DECL LDAT LCPDATP175={VEL 0.1,ACC 100,APO_DIST 5,APO_FAC 50.0,ORI_TYP #VAR,CIRC_TYP #BASE,JERK_FAC 50.0}
DECL FDAT FP175={TOOL_NO 2,BASE_NO 10,IPO_FRAME #BASE,POINT2[] " ",TQ_STATE FALSE}
DECL E6POS XP175={X -116.900,Y -4.570,Z 2.300,A 0.000,B 0.000,C -0.000}
DECL LDAT LCPDATC176={VEL 0.1,ACC 100,APO_DIST 5,APO_FAC 50.0,ORI_TYP #VAR,CIRC_TYP #BASE,JERK_FAC 50.0}
DECL FDAT FC176={TOOL_NO 2,BASE_NO 10,IPO_FRAME #BASE,POINT2[] " ",TQ_STATE FALSE}
DECL E6POS XCAux176={X -55.000,Y 8.590,Z 2.300,A 0.000,B 0.000,C -0.000}
DECL E6POS XCDes176={X 6.900,Y -4.570,Z 2.300,A 0.000,B 0.000,C -0.000}
DECL LDAT LCPDATC177={VEL 0.5,ACC 100,APO_DIST 5,APO_FAC 50.0,ORI_TYP #VAR,CIRC_TYP #BASE,JERK_FAC 50.0}
DECL FDAT FC177={TOOL_NO 2,BASE_NO 10,IPO_FRAME #BASE,POINT2[] " ",TQ_STATE FALSE}
DECL E6POS XCAux177={X 30.100,Y -17.430,Z 2.300,A 0.000,B 0.000,C -0.000}
DECL E6POS XCDes177={X 28.990,Y -19.090,Z 2.300,A 0.000,B 0.000,C -0.000}
DECL LDAT LCPDATP178={VEL 0.1,ACC 100,APO_DIST 5,APO_FAC 50.0,ORI_TYP #VAR,CIRC_TYP #BASE,JERK_FAC 50.0}
DECL FDAT FP178={TOOL_NO 2,BASE_NO 10,IPO_FRAME #BASE,POINT2[] " ",TQ_STATE FALSE}
DECL E6POS XP178={X 6.090,Y -6.390,Z 2.300,A 0.000,B 0.000,C -0.000}
DECL LDAT LCPDATC179={VEL 0.1,ACC 100,APO_DIST 5,APO_FAC 50.0,ORI_TYP #VAR,CIRC_TYP #BASE,JERK_FAC 50.0}
DECL FDAT FC179={TOOL_NO 2,BASE_NO 10,IPO_FRAME #BASE,POINT2[] " ",TQ_STATE FALSE}
DECL E6POS XCAux179={X -55.000,Y 6.590,Z 2.300,A 0.000,B 0.000,C -0.000}
DECL E6POS XCDes179={X -116.090,Y -6.390,Z 2.300,A 0.000,B 0.000,C -0.000}
DECL LDAT LCPDATC180={VEL 0.5,ACC 100,APO_DIST 5,APO_FAC 50.0,ORI_TYP #VAR,CIRC_TYP #BASE,JERK_FAC 50.0}
DECL FDAT FC180={TOOL_NO 2,BASE_NO 10,IPO_FRAME #BASE,POINT2[] " ",TQ_STATE FALSE}
DECL E6POS XCAux180={X -138.990,Y -19.090,Z 2.300,A 0.000,B 0.000,C -0.000}
DECL E6POS XCDes180={X -137.870,Y -20.740,Z 2.300,A 0.000,B 0.000,C -0.000}
DECL LDAT LCPDATP181={VEL 0.1,ACC 100,APO_DIST 5,APO_FAC 50.0,ORI_TYP #VAR,CIRC_TYP #BASE,JERK_FAC 50.0}
DECL FDAT FP181={TOOL_NO 2,BASE_NO 10,IPO_FRAME #BASE,POINT2[] " ",TQ_STATE FALSE}
DECL E6POS XP181={X -115.270,Y -8.220,Z 2.300,A 0.000,B 0.000,C -0.000}
DECL LDAT LCPDATC182={VEL 0.1,ACC 100,APO_DIST 5,APO_FAC 50.0,ORI_TYP #VAR,CIRC_TYP #BASE,JERK_FAC 50.0}
DECL FDAT FC182={TOOL_NO 2,BASE_NO 10,IPO_FRAME #BASE,POINT2[] " ",TQ_STATE FALSE}
DECL E6POS XCAux182={X -55.000,Y 4.590,Z 2.300,A 0.000,B 0.000,C -0.000}
DECL E6POS XCDes182={X 5.270,Y -8.220,Z 2.300,A 0.000,B 0.000,C -0.000}
DECL LDAT LCPDATC183={VEL 0.5,ACC 100,APO_DIST 5,APO_FAC 50.0,ORI_TYP #VAR,CIRC_TYP #BASE,JERK_FAC 50.0}
DECL FDAT FC183={TOOL_NO 2,BASE_NO 10,IPO_FRAME #BASE,POINT2[] " ",TQ_STATE FALSE}
DECL E6POS XCAux183={X 27.870,Y -20.740,Z 2.300,A 0.000,B 0.000,C -0.000}
DECL E6POS XCDes183={X 26.750,Y -22.400,Z 2.300,A 0.000,B 0.000,C -0.000}
DECL LDAT LCPDATP184={VEL 0.1,ACC 100,APO_DIST 5,APO_FAC 50.0,ORI_TYP #VAR,CIRC_TYP #BASE,JERK_FAC 50.0}
DECL FDAT FP184={TOOL_NO 2,BASE_NO 10,IPO_FRAME #BASE,POINT2[] " ",TQ_STATE FALSE}
DECL E6POS XP184={X 4.460,Y -10.050,Z 2.300,A 0.000,B 0.000,C -0.000}
DECL LDAT LCPDATC185={VEL 0.1,ACC 100,APO_DIST 5,APO_FAC 50.0,ORI_TYP #VAR,CIRC_TYP #BASE,JERK_FAC 50.0}
DECL FDAT FC185={TOOL_NO 2,BASE_NO 10,IPO_FRAME #BASE,POINT2[] " ",TQ_STATE FALSE}
DECL E6POS XCAux185={X -55.000,Y 2.590,Z 2.300,A 0.000,B 0.000,C -0.000}
DECL E6POS XCDes185={X -114.460,Y -10.050,Z 2.300,A 0.000,B 0.000,C -0.000}
DECL LDAT LCPDATC186={VEL 0.5,ACC 100,APO_DIST 5,APO_FAC 50.0,ORI_TYP #VAR,CIRC_TYP #BASE,JERK_FAC 50.0}
DECL FDAT FC186={TOOL_NO 2,BASE_NO 10,IPO_FRAME #BASE,POINT2[] " ",TQ_STATE FALSE}
DECL E6POS XCAux186={X -136.750,Y -22.400,Z 2.300,A 0.000,B 0.000,C -0.000}
DECL E6POS XCDes186={X -135.630,Y -24.060,Z 2.300,A 0.000,B 0.000,C -0.000}
DECL LDAT LCPDATP187={VEL 0.1,ACC 100,APO_DIST 5,APO_FAC 50.0,ORI_TYP #VAR,CIRC_TYP #BASE,JERK_FAC 50.0}
DECL FDAT FP187={TOOL_NO 2,BASE_NO 10,IPO_FRAME #BASE,POINT2[] " ",TQ_STATE FALSE}
DECL E6POS XP187={X -113.650,Y -11.880,Z 2.300,A 0.000,B 0.000,C -0.000}
DECL LDAT LCPDATC188={VEL 0.1,ACC 100,APO_DIST 5,APO_FAC 50.0,ORI_TYP #VAR,CIRC_TYP #BASE,JERK_FAC 50.0}
DECL FDAT FC188={TOOL_NO 2,BASE_NO 10,IPO_FRAME #BASE,POINT2[] " ",TQ_STATE FALSE}
DECL E6POS XCAux188={X -55.000,Y 0.590,Z 2.300,A 0.000,B 0.000,C -0.000}
DECL E6POS XCDes188={X 3.650,Y -11.880,Z 2.300,A 0.000,B 0.000,C -0.000}
DECL LDAT LCPDATC189={VEL 0.5,ACC 100,APO_DIST 5,APO_FAC 50.0,ORI_TYP #VAR,CIRC_TYP #BASE,JERK_FAC 50.0}
DECL FDAT FC189={TOOL_NO 2,BASE_NO 10,IPO_FRAME #BASE,POINT2[] " ",TQ_STATE FALSE}
DECL E6POS XCAux189={X 25.630,Y -24.060,Z 2.300,A 0.000,B 0.000,C -0.000}
DECL E6POS XCDes189={X 24.510,Y -25.720,Z 2.300,A 0.000,B 0.000,C -0.000}
DECL LDAT LCPDATP190={VEL 0.1,ACC 100,APO_DIST 5,APO_FAC 50.0,ORI_TYP #VAR,CIRC_TYP #BASE,JERK_FAC 50.0}
DECL FDAT FP190={TOOL_NO 2,BASE_NO 10,IPO_FRAME #BASE,POINT2[] " ",TQ_STATE FALSE}
DECL E6POS XP190={X 2.830,Y -13.700,Z 2.300,A 0.000,B 0.000,C -0.000}
DECL LDAT LCPDATC191={VEL 0.1,ACC 100,APO_DIST 5,APO_FAC 50.0,ORI_TYP #VAR,CIRC_TYP #BASE,JERK_FAC 50.0}
DECL FDAT FC191={TOOL_NO 2,BASE_NO 10,IPO_FRAME #BASE,POINT2[] " ",TQ_STATE FALSE}
DECL E6POS XCAux191={X -55.000,Y -1.410,Z 2.300,A 0.000,B 0.000,C -0.000}
DECL E6POS XCDes191={X -112.830,Y -13.700,Z 2.300,A 0.000,B 0.000,C -0.000}
DECL LDAT LCPDATC192={VEL 0.5,ACC 100,APO_DIST 5,APO_FAC 50.0,ORI_TYP #VAR,CIRC_TYP #BASE,JERK_FAC 50.0}
DECL FDAT FC192={TOOL_NO 2,BASE_NO 10,IPO_FRAME #BASE,POINT2[] " ",TQ_STATE FALSE}
DECL E6POS XCAux192={X -134.510,Y -25.720,Z 2.300,A 0.000,B 0.000,C -0.000}
DECL E6POS XCDes192={X -133.390,Y -27.380,Z 2.300,A 0.000,B 0.000,C -0.000}
DECL LDAT LCPDATP193={VEL 0.1,ACC 100,APO_DIST 5,APO_FAC 50.0,ORI_TYP #VAR,CIRC_TYP #BASE,JERK_FAC 50.0}
DECL FDAT FP193={TOOL_NO 2,BASE_NO 10,IPO_FRAME #BASE,POINT2[] " ",TQ_STATE FALSE}
DECL E6POS XP193={X -112.020,Y -15.530,Z 2.300,A 0.000,B 0.000,C -0.000}
DECL LDAT LCPDATC194={VEL 0.1,ACC 100,APO_DIST 5,APO_FAC 50.0,ORI_TYP #VAR,CIRC_TYP #BASE,JERK_FAC 50.0}
DECL FDAT FC194={TOOL_NO 2,BASE_NO 10,IPO_FRAME #BASE,POINT2[] " ",TQ_STATE FALSE}
DECL E6POS XCAux194={X -55.000,Y -3.410,Z 2.300,A 0.000,B 0.000,C -0.000}
DECL E6POS XCDes194={X 2.020,Y -15.530,Z 2.300,A 0.000,B 0.000,C -0.000}
DECL LDAT LCPDATC195={VEL 0.5,ACC 100,APO_DIST 5,APO_FAC 50.0,ORI_TYP #VAR,CIRC_TYP #BASE,JERK_FAC 50.0}
DECL FDAT FC195={TOOL_NO 2,BASE_NO 10,IPO_FRAME #BASE,POINT2[] " ",TQ_STATE FALSE}
DECL E6POS XCAux195={X 23.390,Y -27.380,Z 2.300,A 0.000,B 0.000,C -0.000}
DECL E6POS XCDes195={X 22.270,Y -29.040,Z 2.300,A 0.000,B 0.000,C -0.000}
DECL LDAT LCPDATP196={VEL 0.1,ACC 100,APO_DIST 5,APO_FAC 50.0,ORI_TYP #VAR,CIRC_TYP #BASE,JERK_FAC 50.0}
DECL FDAT FP196={TOOL_NO 2,BASE_NO 10,IPO_FRAME #BASE,POINT2[] " ",TQ_STATE FALSE}
DECL E6POS XP196={X 1.210,Y -17.360,Z 2.300,A 0.000,B 0.000,C -0.000}
DECL LDAT LCPDATC197={VEL 0.1,ACC 100,APO_DIST 5,APO_FAC 50.0,ORI_TYP #VAR,CIRC_TYP #BASE,JERK_FAC 50.0}
DECL FDAT FC197={TOOL_NO 2,BASE_NO 10,IPO_FRAME #BASE,POINT2[] " ",TQ_STATE FALSE}
DECL E6POS XCAux197={X -55.000,Y -5.410,Z 2.300,A 0.000,B 0.000,C -0.000}
DECL E6POS XCDes197={X -111.210,Y -17.360,Z 2.300,A 0.000,B 0.000,C -0.000}
DECL LDAT LCPDATC198={VEL 0.5,ACC 100,APO_DIST 5,APO_FAC 50.0,ORI_TYP #VAR,CIRC_TYP #BASE,JERK_FAC 50.0}
DECL FDAT FC198={TOOL_NO 2,BASE_NO 10,IPO_FRAME #BASE,POINT2[] " ",TQ_STATE FALSE}
DECL E6POS XCAux198={X -132.270,Y -29.040,Z 2.300,A 0.000,B 0.000,C -0.000}
DECL E6POS XCDes198={X -131.990,Y -29.450,Z 2.300,A -0.000,B -0.040,C -0.060}
DECL LDAT LCPDATP199={VEL 0.1,ACC 100,APO_DIST 5,APO_FAC 50.0,ORI_TYP #VAR,CIRC_TYP #BASE,JERK_FAC 50.0}
DECL FDAT FP199={TOOL_NO 2,BASE_NO 10,IPO_FRAME #BASE,POINT2[] " ",TQ_STATE FALSE}
DECL E6POS XP199={X -111.000,Y -17.820,Z 2.300,A -0.000,B -0.030,C -0.070}
DECL LDAT LCPDATC200={VEL 0.1,ACC 100,APO_DIST 5,APO_FAC 50.0,ORI_TYP #VAR,CIRC_TYP #BASE,JERK_FAC 50.0}
DECL FDAT FC200={TOOL_NO 2,BASE_NO 10,IPO_FRAME #BASE,POINT2[] " ",TQ_STATE FALSE}
DECL E6POS XCAux200={X -55.000,Y -5.920,Z 2.300,A 0.000,B 0.000,C -0.070}
DECL E6POS XCDes200={X 1.000,Y -17.820,Z 2.300,A 0.000,B 0.030,C -0.070}
DECL LDAT LCPDATC201={VEL 0.5,ACC 100,APO_DIST 5,APO_FAC 50.0,ORI_TYP #VAR,CIRC_TYP #BASE,JERK_FAC 50.0}
DECL FDAT FC201={TOOL_NO 2,BASE_NO 10,IPO_FRAME #BASE,POINT2[] " ",TQ_STATE FALSE}
DECL E6POS XCAux201={X 21.990,Y -29.450,Z 2.300,A 0.000,B 0.040,C -0.060}
DECL E6POS XCDes201={X 21.990,Y -29.460,Z 1.900,A 0.000,B 0.030,C -0.040}
DECL LDAT LCPDATP202={VEL 0.1,ACC 100,APO_DIST 5,APO_FAC 50.0,ORI_TYP #VAR,CIRC_TYP #BASE,JERK_FAC 50.0}
DECL FDAT FP202={TOOL_NO 2,BASE_NO 10,IPO_FRAME #BASE,POINT2[] " ",TQ_STATE FALSE}
DECL E6POS XP202={X 1.000,Y -17.820,Z 1.900,A 0.000,B 0.020,C -0.040}
DECL LDAT LCPDATC203={VEL 0.1,ACC 100,APO_DIST 5,APO_FAC 50.0,ORI_TYP #VAR,CIRC_TYP #BASE,JERK_FAC 50.0}
DECL FDAT FC203={TOOL_NO 2,BASE_NO 10,IPO_FRAME #BASE,POINT2[] " ",TQ_STATE FALSE}
DECL E6POS XCAux203={X -55.000,Y -5.920,Z 1.900,A 0.000,B 0.000,C -0.050}
DECL E6POS XCDes203={X -111.000,Y -17.820,Z 1.900,A -0.000,B -0.020,C -0.040}
DECL LDAT LCPDATC204={VEL 0.5,ACC 100,APO_DIST 5,APO_FAC 50.0,ORI_TYP #VAR,CIRC_TYP #BASE,JERK_FAC 50.0}
DECL FDAT FC204={TOOL_NO 2,BASE_NO 10,IPO_FRAME #BASE,POINT2[] " ",TQ_STATE FALSE}
DECL E6POS XCAux204={X -131.990,Y -29.460,Z 1.900,A -0.000,B -0.030,C -0.040}
DECL E6POS XCDes204={X -132.150,Y -29.220,Z 1.900,A 0.000,B 0.000,C -0.000}
DECL LDAT LCPDATP205={VEL 0.1,ACC 100,APO_DIST 5,APO_FAC 50.0,ORI_TYP #VAR,CIRC_TYP #BASE,JERK_FAC 50.0}
DECL FDAT FP205={TOOL_NO 2,BASE_NO 10,IPO_FRAME #BASE,POINT2[] " ",TQ_STATE FALSE}
DECL E6POS XP205={X -111.120,Y -17.560,Z 1.900,A 0.000,B 0.000,C -0.000}
DECL LDAT LCPDATC206={VEL 0.1,ACC 100,APO_DIST 5,APO_FAC 50.0,ORI_TYP #VAR,CIRC_TYP #BASE,JERK_FAC 50.0}
DECL FDAT FC206={TOOL_NO 2,BASE_NO 10,IPO_FRAME #BASE,POINT2[] " ",TQ_STATE FALSE}
DECL E6POS XCAux206={X -55.000,Y -5.630,Z 1.900,A 0.000,B 0.000,C -0.000}
DECL E6POS XCDes206={X 1.120,Y -17.560,Z 1.900,A 0.000,B 0.000,C -0.000}
DECL LDAT LCPDATC207={VEL 0.5,ACC 100,APO_DIST 5,APO_FAC 50.0,ORI_TYP #VAR,CIRC_TYP #BASE,JERK_FAC 50.0}
DECL FDAT FC207={TOOL_NO 2,BASE_NO 10,IPO_FRAME #BASE,POINT2[] " ",TQ_STATE FALSE}
DECL E6POS XCAux207={X 22.150,Y -29.220,Z 1.900,A 0.000,B 0.000,C -0.000}
DECL E6POS XCDes207={X 23.270,Y -27.560,Z 1.900,A 0.000,B 0.000,C -0.000}
DECL LDAT LCPDATP208={VEL 0.1,ACC 100,APO_DIST 5,APO_FAC 50.0,ORI_TYP #VAR,CIRC_TYP #BASE,JERK_FAC 50.0}
DECL FDAT FP208={TOOL_NO 2,BASE_NO 10,IPO_FRAME #BASE,POINT2[] " ",TQ_STATE FALSE}
DECL E6POS XP208={X 1.930,Y -15.730,Z 1.900,A 0.000,B 0.000,C -0.000}
DECL LDAT LCPDATC209={VEL 0.1,ACC 100,APO_DIST 5,APO_FAC 50.0,ORI_TYP #VAR,CIRC_TYP #BASE,JERK_FAC 50.0}
DECL FDAT FC209={TOOL_NO 2,BASE_NO 10,IPO_FRAME #BASE,POINT2[] " ",TQ_STATE FALSE}
DECL E6POS XCAux209={X -55.000,Y -3.630,Z 1.900,A 0.000,B 0.000,C -0.000}
DECL E6POS XCDes209={X -111.930,Y -15.730,Z 1.900,A 0.000,B 0.000,C -0.000}
DECL LDAT LCPDATC210={VEL 0.5,ACC 100,APO_DIST 5,APO_FAC 50.0,ORI_TYP #VAR,CIRC_TYP #BASE,JERK_FAC 50.0}
DECL FDAT FC210={TOOL_NO 2,BASE_NO 10,IPO_FRAME #BASE,POINT2[] " ",TQ_STATE FALSE}
DECL E6POS XCAux210={X -133.270,Y -27.560,Z 1.900,A 0.000,B 0.000,C -0.000}
DECL E6POS XCDes210={X -134.390,Y -25.900,Z 1.900,A 0.000,B 0.000,C -0.000}
DECL LDAT LCPDATP211={VEL 0.1,ACC 100,APO_DIST 5,APO_FAC 50.0,ORI_TYP #VAR,CIRC_TYP #BASE,JERK_FAC 50.0}
DECL FDAT FP211={TOOL_NO 2,BASE_NO 10,IPO_FRAME #BASE,POINT2[] " ",TQ_STATE FALSE}
DECL E6POS XP211={X -112.750,Y -13.900,Z 1.900,A 0.000,B 0.000,C -0.000}
DECL LDAT LCPDATC212={VEL 0.1,ACC 100,APO_DIST 5,APO_FAC 50.0,ORI_TYP #VAR,CIRC_TYP #BASE,JERK_FAC 50.0}
DECL FDAT FC212={TOOL_NO 2,BASE_NO 10,IPO_FRAME #BASE,POINT2[] " ",TQ_STATE FALSE}
DECL E6POS XCAux212={X -55.000,Y -1.630,Z 1.900,A 0.000,B 0.000,C -0.000}
DECL E6POS XCDes212={X 2.750,Y -13.900,Z 1.900,A 0.000,B 0.000,C -0.000}
DECL LDAT LCPDATC213={VEL 0.5,ACC 100,APO_DIST 5,APO_FAC 50.0,ORI_TYP #VAR,CIRC_TYP #BASE,JERK_FAC 50.0}
DECL FDAT FC213={TOOL_NO 2,BASE_NO 10,IPO_FRAME #BASE,POINT2[] " ",TQ_STATE FALSE}
DECL E6POS XCAux213={X 24.390,Y -25.900,Z 1.900,A 0.000,B 0.000,C -0.000}
DECL E6POS XCDes213={X 25.510,Y -24.240,Z 1.900,A 0.000,B 0.000,C -0.000}
DECL LDAT LCPDATP214={VEL 0.1,ACC 100,APO_DIST 5,APO_FAC 50.0,ORI_TYP #VAR,CIRC_TYP #BASE,JERK_FAC 50.0}
DECL FDAT FP214={TOOL_NO 2,BASE_NO 10,IPO_FRAME #BASE,POINT2[] " ",TQ_STATE FALSE}
DECL E6POS XP214={X 3.560,Y -12.080,Z 1.900,A 0.000,B 0.000,C -0.000}
DECL LDAT LCPDATC215={VEL 0.1,ACC 100,APO_DIST 5,APO_FAC 50.0,ORI_TYP #VAR,CIRC_TYP #BASE,JERK_FAC 50.0}
DECL FDAT FC215={TOOL_NO 2,BASE_NO 10,IPO_FRAME #BASE,POINT2[] " ",TQ_STATE FALSE}
DECL E6POS XCAux215={X -55.000,Y 0.370,Z 1.900,A 0.000,B 0.000,C -0.000}
DECL E6POS XCDes215={X -113.560,Y -12.080,Z 1.900,A 0.000,B 0.000,C -0.000}
DECL LDAT LCPDATC216={VEL 0.5,ACC 100,APO_DIST 5,APO_FAC 50.0,ORI_TYP #VAR,CIRC_TYP #BASE,JERK_FAC 50.0}
DECL FDAT FC216={TOOL_NO 2,BASE_NO 10,IPO_FRAME #BASE,POINT2[] " ",TQ_STATE FALSE}
DECL E6POS XCAux216={X -135.510,Y -24.240,Z 1.900,A 0.000,B 0.000,C -0.000}
DECL E6POS XCDes216={X -136.630,Y -22.580,Z 1.900,A 0.000,B 0.000,C -0.000}
DECL LDAT LCPDATP217={VEL 0.1,ACC 100,APO_DIST 5,APO_FAC 50.0,ORI_TYP #VAR,CIRC_TYP #BASE,JERK_FAC 50.0}
DECL FDAT FP217={TOOL_NO 2,BASE_NO 10,IPO_FRAME #BASE,POINT2[] " ",TQ_STATE FALSE}
DECL E6POS XP217={X -114.370,Y -10.250,Z 1.900,A 0.000,B 0.000,C -0.000}
DECL LDAT LCPDATC218={VEL 0.1,ACC 100,APO_DIST 5,APO_FAC 50.0,ORI_TYP #VAR,CIRC_TYP #BASE,JERK_FAC 50.0}
DECL FDAT FC218={TOOL_NO 2,BASE_NO 10,IPO_FRAME #BASE,POINT2[] " ",TQ_STATE FALSE}
DECL E6POS XCAux218={X -55.000,Y 2.370,Z 1.900,A 0.000,B 0.000,C -0.000}
DECL E6POS XCDes218={X 4.370,Y -10.250,Z 1.900,A 0.000,B 0.000,C -0.000}
DECL LDAT LCPDATC219={VEL 0.5,ACC 100,APO_DIST 5,APO_FAC 50.0,ORI_TYP #VAR,CIRC_TYP #BASE,JERK_FAC 50.0}
DECL FDAT FC219={TOOL_NO 2,BASE_NO 10,IPO_FRAME #BASE,POINT2[] " ",TQ_STATE FALSE}
DECL E6POS XCAux219={X 26.630,Y -22.580,Z 1.900,A 0.000,B 0.000,C -0.000}
DECL E6POS XCDes219={X 27.740,Y -20.930,Z 1.900,A 0.000,B 0.000,C -0.000}
DECL LDAT LCPDATP220={VEL 0.1,ACC 100,APO_DIST 5,APO_FAC 50.0,ORI_TYP #VAR,CIRC_TYP #BASE,JERK_FAC 50.0}
DECL FDAT FP220={TOOL_NO 2,BASE_NO 10,IPO_FRAME #BASE,POINT2[] " ",TQ_STATE FALSE}
DECL E6POS XP220={X 5.190,Y -8.420,Z 1.900,A 0.000,B 0.000,C -0.000}
DECL LDAT LCPDATC221={VEL 0.1,ACC 100,APO_DIST 5,APO_FAC 50.0,ORI_TYP #VAR,CIRC_TYP #BASE,JERK_FAC 50.0}
DECL FDAT FC221={TOOL_NO 2,BASE_NO 10,IPO_FRAME #BASE,POINT2[] " ",TQ_STATE FALSE}
DECL E6POS XCAux221={X -55.000,Y 4.370,Z 1.900,A 0.000,B 0.000,C -0.000}
DECL E6POS XCDes221={X -115.190,Y -8.420,Z 1.900,A 0.000,B 0.000,C -0.000}
DECL LDAT LCPDATC222={VEL 0.5,ACC 100,APO_DIST 5,APO_FAC 50.0,ORI_TYP #VAR,CIRC_TYP #BASE,JERK_FAC 50.0}
DECL FDAT FC222={TOOL_NO 2,BASE_NO 10,IPO_FRAME #BASE,POINT2[] " ",TQ_STATE FALSE}
DECL E6POS XCAux222={X -137.740,Y -20.930,Z 1.900,A 0.000,B 0.000,C -0.000}
DECL E6POS XCDes222={X -138.860,Y -19.270,Z 1.900,A 0.000,B 0.000,C -0.000}
DECL LDAT LCPDATP223={VEL 0.1,ACC 100,APO_DIST 5,APO_FAC 50.0,ORI_TYP #VAR,CIRC_TYP #BASE,JERK_FAC 50.0}
DECL FDAT FP223={TOOL_NO 2,BASE_NO 10,IPO_FRAME #BASE,POINT2[] " ",TQ_STATE FALSE}
DECL E6POS XP223={X -116.000,Y -6.590,Z 1.900,A 0.000,B 0.000,C -0.000}
DECL LDAT LCPDATC224={VEL 0.1,ACC 100,APO_DIST 5,APO_FAC 50.0,ORI_TYP #VAR,CIRC_TYP #BASE,JERK_FAC 50.0}
DECL FDAT FC224={TOOL_NO 2,BASE_NO 10,IPO_FRAME #BASE,POINT2[] " ",TQ_STATE FALSE}
DECL E6POS XCAux224={X -55.000,Y 6.370,Z 1.900,A 0.000,B 0.000,C -0.000}
DECL E6POS XCDes224={X 6.000,Y -6.590,Z 1.900,A 0.000,B 0.000,C -0.000}
DECL LDAT LCPDATC225={VEL 0.5,ACC 100,APO_DIST 5,APO_FAC 50.0,ORI_TYP #VAR,CIRC_TYP #BASE,JERK_FAC 50.0}
DECL FDAT FC225={TOOL_NO 2,BASE_NO 10,IPO_FRAME #BASE,POINT2[] " ",TQ_STATE FALSE}
DECL E6POS XCAux225={X 28.860,Y -19.270,Z 1.900,A 0.000,B 0.000,C -0.000}
DECL E6POS XCDes225={X 29.980,Y -17.610,Z 1.900,A 0.000,B 0.000,C -0.000}
DECL LDAT LCPDATP226={VEL 0.1,ACC 100,APO_DIST 5,APO_FAC 50.0,ORI_TYP #VAR,CIRC_TYP #BASE,JERK_FAC 50.0}
DECL FDAT FP226={TOOL_NO 2,BASE_NO 10,IPO_FRAME #BASE,POINT2[] " ",TQ_STATE FALSE}
DECL E6POS XP226={X 6.810,Y -4.770,Z 1.900,A 0.000,B 0.000,C -0.000}
DECL LDAT LCPDATC227={VEL 0.1,ACC 100,APO_DIST 5,APO_FAC 50.0,ORI_TYP #VAR,CIRC_TYP #BASE,JERK_FAC 50.0}
DECL FDAT FC227={TOOL_NO 2,BASE_NO 10,IPO_FRAME #BASE,POINT2[] " ",TQ_STATE FALSE}
DECL E6POS XCAux227={X -55.000,Y 8.370,Z 1.900,A 0.000,B 0.000,C -0.000}
DECL E6POS XCDes227={X -116.810,Y -4.770,Z 1.900,A 0.000,B 0.000,C -0.000}
DECL LDAT LCPDATC228={VEL 0.5,ACC 100,APO_DIST 5,APO_FAC 50.0,ORI_TYP #VAR,CIRC_TYP #BASE,JERK_FAC 50.0}
DECL FDAT FC228={TOOL_NO 2,BASE_NO 10,IPO_FRAME #BASE,POINT2[] " ",TQ_STATE FALSE}
DECL E6POS XCAux228={X -139.980,Y -17.610,Z 1.900,A 0.000,B 0.000,C -0.000}
DECL E6POS XCDes228={X -141.100,Y -15.950,Z 1.900,A 0.000,B 0.000,C -0.000}
DECL LDAT LCPDATP229={VEL 0.1,ACC 100,APO_DIST 5,APO_FAC 50.0,ORI_TYP #VAR,CIRC_TYP #BASE,JERK_FAC 50.0}
DECL FDAT FP229={TOOL_NO 2,BASE_NO 10,IPO_FRAME #BASE,POINT2[] " ",TQ_STATE FALSE}
DECL E6POS XP229={X -117.630,Y -2.940,Z 1.900,A 0.000,B 0.000,C -0.000}
DECL LDAT LCPDATC230={VEL 0.1,ACC 100,APO_DIST 5,APO_FAC 50.0,ORI_TYP #VAR,CIRC_TYP #BASE,JERK_FAC 50.0}
DECL FDAT FC230={TOOL_NO 2,BASE_NO 10,IPO_FRAME #BASE,POINT2[] " ",TQ_STATE FALSE}
DECL E6POS XCAux230={X -55.000,Y 10.370,Z 1.900,A 0.000,B 0.000,C -0.000}
DECL E6POS XCDes230={X 7.630,Y -2.940,Z 1.900,A 0.000,B 0.000,C -0.000}
DECL LDAT LCPDATC231={VEL 0.5,ACC 100,APO_DIST 5,APO_FAC 50.0,ORI_TYP #VAR,CIRC_TYP #BASE,JERK_FAC 50.0}
DECL FDAT FC231={TOOL_NO 2,BASE_NO 10,IPO_FRAME #BASE,POINT2[] " ",TQ_STATE FALSE}
DECL E6POS XCAux231={X 31.100,Y -15.950,Z 1.900,A 0.000,B 0.000,C -0.000}
DECL E6POS XCDes231={X 31.090,Y -15.970,Z 1.690,A 0.000,B 8.070,C -12.130}
DECL LDAT LCPDATP232={VEL 0.1,ACC 100,APO_DIST 5,APO_FAC 50.0,ORI_TYP #VAR,CIRC_TYP #BASE,JERK_FAC 50.0}
DECL FDAT FP232={TOOL_NO 2,BASE_NO 10,IPO_FRAME #BASE,POINT2[] " ",TQ_STATE FALSE}
DECL E6POS XP232={X 7.620,Y -2.960,Z 1.690,A 0.000,B 5.860,C -13.330}
DECL LDAT LCPDATC233={VEL 0.1,ACC 100,APO_DIST 5,APO_FAC 50.0,ORI_TYP #VAR,CIRC_TYP #BASE,JERK_FAC 50.0}
DECL FDAT FC233={TOOL_NO 2,BASE_NO 10,IPO_FRAME #BASE,POINT2[] " ",TQ_STATE FALSE}
DECL E6POS XCAux233={X -55.000,Y 10.350,Z 1.690,A 0.000,B 0.000,C -14.540}
DECL E6POS XCDes233={X -117.620,Y -2.960,Z 1.690,A -0.000,B -5.860,C -13.330}
DECL LDAT LCPDATC234={VEL 0.5,ACC 100,APO_DIST 5,APO_FAC 50.0,ORI_TYP #VAR,CIRC_TYP #BASE,JERK_FAC 50.0}
DECL FDAT FC234={TOOL_NO 2,BASE_NO 10,IPO_FRAME #BASE,POINT2[] " ",TQ_STATE FALSE}
DECL E6POS XCAux234={X -141.090,Y -15.970,Z 1.690,A -0.000,B -8.070,C -12.130}
DECL E6POS XCDes234={X -140.960,Y -16.150,Z 1.330,A -0.000,B -7.450,C -11.170}
DECL LDAT LCPDATP235={VEL 0.1,ACC 100,APO_DIST 5,APO_FAC 50.0,ORI_TYP #VAR,CIRC_TYP #BASE,JERK_FAC 50.0}
DECL FDAT FP235={TOOL_NO 2,BASE_NO 10,IPO_FRAME #BASE,POINT2[] " ",TQ_STATE FALSE}
DECL E6POS XP235={X -117.530,Y -3.160,Z 1.330,A -0.000,B -5.410,C -12.280}
DECL LDAT LCPDATC236={VEL 0.1,ACC 100,APO_DIST 5,APO_FAC 50.0,ORI_TYP #VAR,CIRC_TYP #BASE,JERK_FAC 50.0}
DECL FDAT FC236={TOOL_NO 2,BASE_NO 10,IPO_FRAME #BASE,POINT2[] " ",TQ_STATE FALSE}
DECL E6POS XCAux236={X -55.000,Y 10.130,Z 1.330,A 0.000,B 0.000,C -13.400}
DECL E6POS XCDes236={X 7.530,Y -3.160,Z 1.330,A 0.000,B 5.410,C -12.280}
DECL LDAT LCPDATC237={VEL 0.5,ACC 100,APO_DIST 5,APO_FAC 50.0,ORI_TYP #VAR,CIRC_TYP #BASE,JERK_FAC 50.0}
DECL FDAT FC237={TOOL_NO 2,BASE_NO 10,IPO_FRAME #BASE,POINT2[] " ",TQ_STATE FALSE}
DECL E6POS XCAux237={X 30.960,Y -16.150,Z 1.330,A 0.000,B 7.450,C -11.170}
DECL E6POS XCDes237={X 30.980,Y -16.130,Z 1.500,A 0.000,B 0.000,C -0.000}
DECL LDAT LCPDATP238={VEL 0.1,ACC 100,APO_DIST 5,APO_FAC 50.0,ORI_TYP #VAR,CIRC_TYP #BASE,JERK_FAC 50.0}
DECL FDAT FP238={TOOL_NO 2,BASE_NO 10,IPO_FRAME #BASE,POINT2[] " ",TQ_STATE FALSE}
DECL E6POS XP238={X 7.540,Y -3.140,Z 1.500,A 0.000,B 0.000,C -0.000}
DECL LDAT LCPDATC239={VEL 0.1,ACC 100,APO_DIST 5,APO_FAC 50.0,ORI_TYP #VAR,CIRC_TYP #BASE,JERK_FAC 50.0}
DECL FDAT FC239={TOOL_NO 2,BASE_NO 10,IPO_FRAME #BASE,POINT2[] " ",TQ_STATE FALSE}
DECL E6POS XCAux239={X -55.000,Y 10.150,Z 1.500,A 0.000,B 0.000,C -0.000}
DECL E6POS XCDes239={X -117.540,Y -3.140,Z 1.500,A 0.000,B 0.000,C -0.000}
DECL LDAT LCPDATC240={VEL 0.5,ACC 100,APO_DIST 5,APO_FAC 50.0,ORI_TYP #VAR,CIRC_TYP #BASE,JERK_FAC 50.0}
DECL FDAT FC240={TOOL_NO 2,BASE_NO 10,IPO_FRAME #BASE,POINT2[] " ",TQ_STATE FALSE}
DECL E6POS XCAux240={X -140.980,Y -16.130,Z 1.500,A 0.000,B 0.000,C -0.000}
DECL E6POS XCDes240={X -139.860,Y -17.790,Z 1.500,A 0.000,B 0.000,C -0.000}
DECL LDAT LCPDATP241={VEL 0.1,ACC 100,APO_DIST 5,APO_FAC 50.0,ORI_TYP #VAR,CIRC_TYP #BASE,JERK_FAC 50.0}
DECL FDAT FP241={TOOL_NO 2,BASE_NO 10,IPO_FRAME #BASE,POINT2[] " ",TQ_STATE FALSE}
DECL E6POS XP241={X -116.720,Y -4.970,Z 1.500,A 0.000,B 0.000,C -0.000}
DECL LDAT LCPDATC242={VEL 0.1,ACC 100,APO_DIST 5,APO_FAC 50.0,ORI_TYP #VAR,CIRC_TYP #BASE,JERK_FAC 50.0}
DECL FDAT FC242={TOOL_NO 2,BASE_NO 10,IPO_FRAME #BASE,POINT2[] " ",TQ_STATE FALSE}
DECL E6POS XCAux242={X -55.000,Y 8.150,Z 1.500,A 0.000,B 0.000,C -0.000}
DECL E6POS XCDes242={X 6.720,Y -4.970,Z 1.500,A 0.000,B 0.000,C -0.000}
DECL LDAT LCPDATC243={VEL 0.5,ACC 100,APO_DIST 5,APO_FAC 50.0,ORI_TYP #VAR,CIRC_TYP #BASE,JERK_FAC 50.0}
DECL FDAT FC243={TOOL_NO 2,BASE_NO 10,IPO_FRAME #BASE,POINT2[] " ",TQ_STATE FALSE}
DECL E6POS XCAux243={X 29.860,Y -17.790,Z 1.500,A 0.000,B 0.000,C -0.000}
DECL E6POS XCDes243={X 28.740,Y -19.450,Z 1.500,A 0.000,B 0.000,C -0.000}
DECL LDAT LCPDATP244={VEL 0.1,ACC 100,APO_DIST 5,APO_FAC 50.0,ORI_TYP #VAR,CIRC_TYP #BASE,JERK_FAC 50.0}
DECL FDAT FP244={TOOL_NO 2,BASE_NO 10,IPO_FRAME #BASE,POINT2[] " ",TQ_STATE FALSE}
DECL E6POS XP244={X 5.910,Y -6.790,Z 1.500,A 0.000,B 0.000,C -0.000}
DECL LDAT LCPDATC245={VEL 0.1,ACC 100,APO_DIST 5,APO_FAC 50.0,ORI_TYP #VAR,CIRC_TYP #BASE,JERK_FAC 50.0}
DECL FDAT FC245={TOOL_NO 2,BASE_NO 10,IPO_FRAME #BASE,POINT2[] " ",TQ_STATE FALSE}
DECL E6POS XCAux245={X -55.000,Y 6.150,Z 1.500,A 0.000,B 0.000,C -0.000}
DECL E6POS XCDes245={X -115.910,Y -6.790,Z 1.500,A 0.000,B 0.000,C -0.000}
DECL LDAT LCPDATC246={VEL 0.5,ACC 100,APO_DIST 5,APO_FAC 50.0,ORI_TYP #VAR,CIRC_TYP #BASE,JERK_FAC 50.0}
DECL FDAT FC246={TOOL_NO 2,BASE_NO 10,IPO_FRAME #BASE,POINT2[] " ",TQ_STATE FALSE}
DECL E6POS XCAux246={X -138.740,Y -19.450,Z 1.500,A 0.000,B 0.000,C -0.000}
DECL E6POS XCDes246={X -137.620,Y -21.110,Z 1.500,A 0.000,B 0.000,C -0.000}
DECL LDAT LCPDATP247={VEL 0.1,ACC 100,APO_DIST 5,APO_FAC 50.0,ORI_TYP #VAR,CIRC_TYP #BASE,JERK_FAC 50.0}
DECL FDAT FP247={TOOL_NO 2,BASE_NO 10,IPO_FRAME #BASE,POINT2[] " ",TQ_STATE FALSE}
DECL E6POS XP247={X -115.100,Y -8.620,Z 1.500,A 0.000,B 0.000,C -0.000}
DECL LDAT LCPDATC248={VEL 0.1,ACC 100,APO_DIST 5,APO_FAC 50.0,ORI_TYP #VAR,CIRC_TYP #BASE,JERK_FAC 50.0}
DECL FDAT FC248={TOOL_NO 2,BASE_NO 10,IPO_FRAME #BASE,POINT2[] " ",TQ_STATE FALSE}
DECL E6POS XCAux248={X -55.000,Y 4.150,Z 1.500,A 0.000,B 0.000,C -0.000}
DECL E6POS XCDes248={X 5.100,Y -8.620,Z 1.500,A 0.000,B 0.000,C -0.000}
DECL LDAT LCPDATC249={VEL 0.5,ACC 100,APO_DIST 5,APO_FAC 50.0,ORI_TYP #VAR,CIRC_TYP #BASE,JERK_FAC 50.0}
DECL FDAT FC249={TOOL_NO 2,BASE_NO 10,IPO_FRAME #BASE,POINT2[] " ",TQ_STATE FALSE}
DECL E6POS XCAux249={X 27.620,Y -21.110,Z 1.500,A 0.000,B 0.000,C -0.000}
DECL E6POS XCDes249={X 26.500,Y -22.770,Z 1.500,A 0.000,B 0.000,C -0.000}
DECL LDAT LCPDATP250={VEL 0.1,ACC 100,APO_DIST 5,APO_FAC 50.0,ORI_TYP #VAR,CIRC_TYP #BASE,JERK_FAC 50.0}
DECL FDAT FP250={TOOL_NO 2,BASE_NO 10,IPO_FRAME #BASE,POINT2[] " ",TQ_STATE FALSE}
DECL E6POS XP250={X 4.280,Y -10.450,Z 1.500,A 0.000,B 0.000,C -0.000}
DECL LDAT LCPDATC251={VEL 0.1,ACC 100,APO_DIST 5,APO_FAC 50.0,ORI_TYP #VAR,CIRC_TYP #BASE,JERK_FAC 50.0}
DECL FDAT FC251={TOOL_NO 2,BASE_NO 10,IPO_FRAME #BASE,POINT2[] " ",TQ_STATE FALSE}
DECL E6POS XCAux251={X -55.000,Y 2.150,Z 1.500,A 0.000,B 0.000,C -0.000}
DECL E6POS XCDes251={X -114.280,Y -10.450,Z 1.500,A 0.000,B 0.000,C -0.000}
DECL LDAT LCPDATC252={VEL 0.5,ACC 100,APO_DIST 5,APO_FAC 50.0,ORI_TYP #VAR,CIRC_TYP #BASE,JERK_FAC 50.0}
DECL FDAT FC252={TOOL_NO 2,BASE_NO 10,IPO_FRAME #BASE,POINT2[] " ",TQ_STATE FALSE}
DECL E6POS XCAux252={X -136.500,Y -22.770,Z 1.500,A 0.000,B 0.000,C -0.000}
DECL E6POS XCDes252={X -135.390,Y -24.420,Z 1.500,A 0.000,B 0.000,C -0.000}
DECL LDAT LCPDATP253={VEL 0.1,ACC 100,APO_DIST 5,APO_FAC 50.0,ORI_TYP #VAR,CIRC_TYP #BASE,JERK_FAC 50.0}
DECL FDAT FP253={TOOL_NO 2,BASE_NO 10,IPO_FRAME #BASE,POINT2[] " ",TQ_STATE FALSE}
DECL E6POS XP253={X -113.470,Y -12.270,Z 1.500,A 0.000,B 0.000,C -0.000}
DECL LDAT LCPDATC254={VEL 0.1,ACC 100,APO_DIST 5,APO_FAC 50.0,ORI_TYP #VAR,CIRC_TYP #BASE,JERK_FAC 50.0}
DECL FDAT FC254={TOOL_NO 2,BASE_NO 10,IPO_FRAME #BASE,POINT2[] " ",TQ_STATE FALSE}
DECL E6POS XCAux254={X -55.000,Y 0.150,Z 1.500,A 0.000,B 0.000,C -0.000}
DECL E6POS XCDes254={X 3.470,Y -12.270,Z 1.500,A 0.000,B 0.000,C -0.000}
DECL LDAT LCPDATC255={VEL 0.5,ACC 100,APO_DIST 5,APO_FAC 50.0,ORI_TYP #VAR,CIRC_TYP #BASE,JERK_FAC 50.0}
DECL FDAT FC255={TOOL_NO 2,BASE_NO 10,IPO_FRAME #BASE,POINT2[] " ",TQ_STATE FALSE}
DECL E6POS XCAux255={X 25.390,Y -24.420,Z 1.500,A 0.000,B 0.000,C -0.000}
DECL E6POS XCDes255={X 24.270,Y -26.080,Z 1.500,A 0.000,B 0.000,C -0.000}
DECL LDAT LCPDATP256={VEL 0.1,ACC 100,APO_DIST 5,APO_FAC 50.0,ORI_TYP #VAR,CIRC_TYP #BASE,JERK_FAC 50.0}
DECL FDAT FP256={TOOL_NO 2,BASE_NO 10,IPO_FRAME #BASE,POINT2[] " ",TQ_STATE FALSE}
DECL E6POS XP256={X 2.660,Y -14.100,Z 1.500,A 0.000,B 0.000,C -0.000}
DECL LDAT LCPDATC257={VEL 0.1,ACC 100,APO_DIST 5,APO_FAC 50.0,ORI_TYP #VAR,CIRC_TYP #BASE,JERK_FAC 50.0}
DECL FDAT FC257={TOOL_NO 2,BASE_NO 10,IPO_FRAME #BASE,POINT2[] " ",TQ_STATE FALSE}
DECL E6POS XCAux257={X -55.000,Y -1.850,Z 1.500,A 0.000,B 0.000,C -0.000}
DECL E6POS XCDes257={X -112.660,Y -14.100,Z 1.500,A 0.000,B 0.000,C -0.000}
DECL LDAT LCPDATC258={VEL 0.5,ACC 100,APO_DIST 5,APO_FAC 50.0,ORI_TYP #VAR,CIRC_TYP #BASE,JERK_FAC 50.0}
DECL FDAT FC258={TOOL_NO 2,BASE_NO 10,IPO_FRAME #BASE,POINT2[] " ",TQ_STATE FALSE}
DECL E6POS XCAux258={X -134.270,Y -26.080,Z 1.500,A 0.000,B 0.000,C -0.000}
DECL E6POS XCDes258={X -133.150,Y -27.740,Z 1.500,A 0.000,B 0.000,C -0.000}
DECL LDAT LCPDATP259={VEL 0.1,ACC 100,APO_DIST 5,APO_FAC 50.0,ORI_TYP #VAR,CIRC_TYP #BASE,JERK_FAC 50.0}
DECL FDAT FP259={TOOL_NO 2,BASE_NO 10,IPO_FRAME #BASE,POINT2[] " ",TQ_STATE FALSE}
DECL E6POS XP259={X -111.840,Y -15.930,Z 1.500,A 0.000,B 0.000,C -0.000}
DECL LDAT LCPDATC260={VEL 0.1,ACC 100,APO_DIST 5,APO_FAC 50.0,ORI_TYP #VAR,CIRC_TYP #BASE,JERK_FAC 50.0}
DECL FDAT FC260={TOOL_NO 2,BASE_NO 10,IPO_FRAME #BASE,POINT2[] " ",TQ_STATE FALSE}
DECL E6POS XCAux260={X -55.000,Y -3.850,Z 1.500,A 0.000,B 0.000,C -0.000}
DECL E6POS XCDes260={X 1.840,Y -15.930,Z 1.500,A 0.000,B 0.000,C -0.000}
DECL LDAT LCPDATC261={VEL 0.5,ACC 100,APO_DIST 5,APO_FAC 50.0,ORI_TYP #VAR,CIRC_TYP #BASE,JERK_FAC 50.0}
DECL FDAT FC261={TOOL_NO 2,BASE_NO 10,IPO_FRAME #BASE,POINT2[] " ",TQ_STATE FALSE}
DECL E6POS XCAux261={X 23.150,Y -27.740,Z 1.500,A 0.000,B 0.000,C -0.000}
DECL E6POS XCDes261={X 22.030,Y -29.400,Z 1.500,A 0.000,B 0.000,C -0.000}
DECL LDAT LCPDATP262={VEL 0.1,ACC 100,APO_DIST 5,APO_FAC 50.0,ORI_TYP #VAR,CIRC_TYP #BASE,JERK_FAC 50.0}
DECL FDAT FP262={TOOL_NO 2,BASE_NO 10,IPO_FRAME #BASE,POINT2[] " ",TQ_STATE FALSE}
DECL E6POS XP262={X 1.030,Y -17.760,Z 1.500,A 0.000,B 0.000,C -0.000}
DECL LDAT LCPDATC263={VEL 0.1,ACC 100,APO_DIST 5,APO_FAC 50.0,ORI_TYP #VAR,CIRC_TYP #BASE,JERK_FAC 50.0}
DECL FDAT FC263={TOOL_NO 2,BASE_NO 10,IPO_FRAME #BASE,POINT2[] " ",TQ_STATE FALSE}
DECL E6POS XCAux263={X -55.000,Y -5.850,Z 1.500,A 0.000,B 0.000,C -0.000}
DECL E6POS XCDes263={X -111.030,Y -17.760,Z 1.500,A 0.000,B 0.000,C -0.000}
DECL LDAT LCPDATC264={VEL 0.5,ACC 100,APO_DIST 5,APO_FAC 50.0,ORI_TYP #VAR,CIRC_TYP #BASE,JERK_FAC 50.0}
DECL FDAT FC264={TOOL_NO 2,BASE_NO 10,IPO_FRAME #BASE,POINT2[] " ",TQ_STATE FALSE}
DECL E6POS XCAux264={X -132.030,Y -29.400,Z 1.500,A 0.000,B 0.000,C -0.000}
DECL E6POS XCDes264={X -131.990,Y -29.460,Z 1.500,A -0.000,B -0.010,C -0.010}
DECL LDAT LCPDATP265={VEL 0.1,ACC 100,APO_DIST 5,APO_FAC 50.0,ORI_TYP #VAR,CIRC_TYP #BASE,JERK_FAC 50.0}
DECL FDAT FP265={TOOL_NO 2,BASE_NO 10,IPO_FRAME #BASE,POINT2[] " ",TQ_STATE FALSE}
DECL E6POS XP265={X -111.000,Y -17.830,Z 1.500,A -0.000,B -0.010,C -0.010}
DECL LDAT LCPDATC266={VEL 0.1,ACC 100,APO_DIST 5,APO_FAC 50.0,ORI_TYP #VAR,CIRC_TYP #BASE,JERK_FAC 50.0}
DECL FDAT FC266={TOOL_NO 2,BASE_NO 10,IPO_FRAME #BASE,POINT2[] " ",TQ_STATE FALSE}
DECL E6POS XCAux266={X -55.000,Y -5.920,Z 1.500,A 0.000,B 0.000,C -0.010}
DECL E6POS XCDes266={X 1.000,Y -17.830,Z 1.500,A 0.000,B 0.010,C -0.010}
DECL LDAT LCPDATC267={VEL 0.5,ACC 100,APO_DIST 5,APO_FAC 50.0,ORI_TYP #VAR,CIRC_TYP #BASE,JERK_FAC 50.0}
DECL FDAT FC267={TOOL_NO 2,BASE_NO 10,IPO_FRAME #BASE,POINT2[] " ",TQ_STATE FALSE}
DECL E6POS XCAux267={X 21.990,Y -29.460,Z 1.500,A 0.000,B 0.010,C -0.010}
DECL E6POS XCDes267={X 22.010,Y -29.440,Z 1.100,A 0.000,B 0.180,C -0.270}
DECL LDAT LCPDATP268={VEL 0.1,ACC 100,APO_DIST 5,APO_FAC 50.0,ORI_TYP #VAR,CIRC_TYP #BASE,JERK_FAC 50.0}
DECL FDAT FP268={TOOL_NO 2,BASE_NO 10,IPO_FRAME #BASE,POINT2[] " ",TQ_STATE FALSE}
DECL E6POS XP268={X 1.010,Y -17.800,Z 1.100,A 0.000,B 0.130,C -0.300}
DECL LDAT LCPDATC269={VEL 0.1,ACC 100,APO_DIST 5,APO_FAC 50.0,ORI_TYP #VAR,CIRC_TYP #BASE,JERK_FAC 50.0}
DECL FDAT FC269={TOOL_NO 2,BASE_NO 10,IPO_FRAME #BASE,POINT2[] " ",TQ_STATE FALSE}
DECL E6POS XCAux269={X -55.000,Y -5.890,Z 1.100,A 0.000,B 0.000,C -0.330}
DECL E6POS XCDes269={X -111.010,Y -17.800,Z 1.100,A -0.000,B -0.130,C -0.300}
DECL LDAT LCPDATC270={VEL 0.5,ACC 100,APO_DIST 5,APO_FAC 50.0,ORI_TYP #VAR,CIRC_TYP #BASE,JERK_FAC 50.0}
DECL FDAT FC270={TOOL_NO 2,BASE_NO 10,IPO_FRAME #BASE,POINT2[] " ",TQ_STATE FALSE}
DECL E6POS XCAux270={X -132.010,Y -29.440,Z 1.100,A -0.000,B -0.180,C -0.270}
DECL E6POS XCDes270={X -133.030,Y -27.920,Z 1.100,A 0.000,B 0.000,C -0.000}
DECL LDAT LCPDATP271={VEL 0.1,ACC 100,APO_DIST 5,APO_FAC 50.0,ORI_TYP #VAR,CIRC_TYP #BASE,JERK_FAC 50.0}
DECL FDAT FP271={TOOL_NO 2,BASE_NO 10,IPO_FRAME #BASE,POINT2[] " ",TQ_STATE FALSE}
DECL E6POS XP271={X -111.750,Y -16.130,Z 1.100,A 0.000,B 0.000,C -0.000}
DECL LDAT LCPDATC272={VEL 0.1,ACC 100,APO_DIST 5,APO_FAC 50.0,ORI_TYP #VAR,CIRC_TYP #BASE,JERK_FAC 50.0}
DECL FDAT FC272={TOOL_NO 2,BASE_NO 10,IPO_FRAME #BASE,POINT2[] " ",TQ_STATE FALSE}
DECL E6POS XCAux272={X -55.000,Y -4.070,Z 1.100,A 0.000,B 0.000,C -0.000}
DECL E6POS XCDes272={X 1.750,Y -16.130,Z 1.100,A 0.000,B 0.000,C -0.000}
DECL LDAT LCPDATC273={VEL 0.5,ACC 100,APO_DIST 5,APO_FAC 50.0,ORI_TYP #VAR,CIRC_TYP #BASE,JERK_FAC 50.0}
DECL FDAT FC273={TOOL_NO 2,BASE_NO 10,IPO_FRAME #BASE,POINT2[] " ",TQ_STATE FALSE}
DECL E6POS XCAux273={X 23.030,Y -27.920,Z 1.100,A 0.000,B 0.000,C -0.000}
DECL E6POS XCDes273={X 24.140,Y -26.260,Z 1.100,A 0.000,B 0.000,C -0.000}
DECL LDAT LCPDATP274={VEL 0.1,ACC 100,APO_DIST 5,APO_FAC 50.0,ORI_TYP #VAR,CIRC_TYP #BASE,JERK_FAC 50.0}
DECL FDAT FP274={TOOL_NO 2,BASE_NO 10,IPO_FRAME #BASE,POINT2[] " ",TQ_STATE FALSE}
DECL E6POS XP274={X 2.570,Y -14.300,Z 1.100,A 0.000,B 0.000,C -0.000}
DECL LDAT LCPDATC275={VEL 0.1,ACC 100,APO_DIST 5,APO_FAC 50.0,ORI_TYP #VAR,CIRC_TYP #BASE,JERK_FAC 50.0}
DECL FDAT FC275={TOOL_NO 2,BASE_NO 10,IPO_FRAME #BASE,POINT2[] " ",TQ_STATE FALSE}
DECL E6POS XCAux275={X -55.000,Y -2.070,Z 1.100,A 0.000,B 0.000,C -0.000}
DECL E6POS XCDes275={X -112.570,Y -14.300,Z 1.100,A 0.000,B 0.000,C -0.000}
DECL LDAT LCPDATC276={VEL 0.5,ACC 100,APO_DIST 5,APO_FAC 50.0,ORI_TYP #VAR,CIRC_TYP #BASE,JERK_FAC 50.0}
DECL FDAT FC276={TOOL_NO 2,BASE_NO 10,IPO_FRAME #BASE,POINT2[] " ",TQ_STATE FALSE}
DECL E6POS XCAux276={X -134.140,Y -26.260,Z 1.100,A 0.000,B 0.000,C -0.000}
DECL E6POS XCDes276={X -135.260,Y -24.610,Z 1.100,A 0.000,B 0.000,C -0.000}
DECL LDAT LCPDATP277={VEL 0.1,ACC 100,APO_DIST 5,APO_FAC 50.0,ORI_TYP #VAR,CIRC_TYP #BASE,JERK_FAC 50.0}
DECL FDAT FP277={TOOL_NO 2,BASE_NO 10,IPO_FRAME #BASE,POINT2[] " ",TQ_STATE FALSE}
DECL E6POS XP277={X -113.380,Y -12.480,Z 1.100,A 0.000,B 0.000,C -0.000}
DECL LDAT LCPDATC278={VEL 0.1,ACC 100,APO_DIST 5,APO_FAC 50.0,ORI_TYP #VAR,CIRC_TYP #BASE,JERK_FAC 50.0}
DECL FDAT FC278={TOOL_NO 2,BASE_NO 10,IPO_FRAME #BASE,POINT2[] " ",TQ_STATE FALSE}
DECL E6POS XCAux278={X -55.000,Y -0.070,Z 1.100,A 0.000,B 0.000,C -0.000}
DECL E6POS XCDes278={X 3.380,Y -12.480,Z 1.100,A 0.000,B 0.000,C -0.000}
DECL LDAT LCPDATC279={VEL 0.5,ACC 100,APO_DIST 5,APO_FAC 50.0,ORI_TYP #VAR,CIRC_TYP #BASE,JERK_FAC 50.0}
DECL FDAT FC279={TOOL_NO 2,BASE_NO 10,IPO_FRAME #BASE,POINT2[] " ",TQ_STATE FALSE}
DECL E6POS XCAux279={X 25.260,Y -24.610,Z 1.100,A 0.000,B 0.000,C -0.000}
DECL E6POS XCDes279={X 26.380,Y -22.950,Z 1.100,A 0.000,B 0.000,C -0.000}
DECL LDAT LCPDATP280={VEL 0.1,ACC 100,APO_DIST 5,APO_FAC 50.0,ORI_TYP #VAR,CIRC_TYP #BASE,JERK_FAC 50.0}
DECL FDAT FP280={TOOL_NO 2,BASE_NO 10,IPO_FRAME #BASE,POINT2[] " ",TQ_STATE FALSE}
DECL E6POS XP280={X 4.190,Y -10.650,Z 1.100,A 0.000,B 0.000,C -0.000}
DECL LDAT LCPDATC281={VEL 0.1,ACC 100,APO_DIST 5,APO_FAC 50.0,ORI_TYP #VAR,CIRC_TYP #BASE,JERK_FAC 50.0}
DECL FDAT FC281={TOOL_NO 2,BASE_NO 10,IPO_FRAME #BASE,POINT2[] " ",TQ_STATE FALSE}
DECL E6POS XCAux281={X -55.000,Y 1.930,Z 1.100,A 0.000,B 0.000,C -0.000}
DECL E6POS XCDes281={X -114.190,Y -10.650,Z 1.100,A 0.000,B 0.000,C -0.000}
DECL LDAT LCPDATC282={VEL 0.5,ACC 100,APO_DIST 5,APO_FAC 50.0,ORI_TYP #VAR,CIRC_TYP #BASE,JERK_FAC 50.0}
DECL FDAT FC282={TOOL_NO 2,BASE_NO 10,IPO_FRAME #BASE,POINT2[] " ",TQ_STATE FALSE}
DECL E6POS XCAux282={X -136.380,Y -22.950,Z 1.100,A 0.000,B 0.000,C -0.000}
DECL E6POS XCDes282={X -137.500,Y -21.290,Z 1.100,A 0.000,B 0.000,C -0.000}
DECL LDAT LCPDATP283={VEL 0.1,ACC 100,APO_DIST 5,APO_FAC 50.0,ORI_TYP #VAR,CIRC_TYP #BASE,JERK_FAC 50.0}
DECL FDAT FP283={TOOL_NO 2,BASE_NO 10,IPO_FRAME #BASE,POINT2[] " ",TQ_STATE FALSE}
DECL E6POS XP283={X -115.010,Y -8.820,Z 1.100,A 0.000,B 0.000,C -0.000}
DECL LDAT LCPDATC284={VEL 0.1,ACC 100,APO_DIST 5,APO_FAC 50.0,ORI_TYP #VAR,CIRC_TYP #BASE,JERK_FAC 50.0}
DECL FDAT FC284={TOOL_NO 2,BASE_NO 10,IPO_FRAME #BASE,POINT2[] " ",TQ_STATE FALSE}
DECL E6POS XCAux284={X -55.000,Y 3.930,Z 1.100,A 0.000,B 0.000,C -0.000}
DECL E6POS XCDes284={X 5.010,Y -8.820,Z 1.100,A 0.000,B 0.000,C -0.000}
DECL LDAT LCPDATC285={VEL 0.5,ACC 100,APO_DIST 5,APO_FAC 50.0,ORI_TYP #VAR,CIRC_TYP #BASE,JERK_FAC 50.0}
DECL FDAT FC285={TOOL_NO 2,BASE_NO 10,IPO_FRAME #BASE,POINT2[] " ",TQ_STATE FALSE}
DECL E6POS XCAux285={X 27.500,Y -21.290,Z 1.100,A 0.000,B 0.000,C -0.000}
DECL E6POS XCDes285={X 28.620,Y -19.630,Z 1.100,A 0.000,B 0.000,C -0.000}
DECL LDAT LCPDATP286={VEL 0.1,ACC 100,APO_DIST 5,APO_FAC 50.0,ORI_TYP #VAR,CIRC_TYP #BASE,JERK_FAC 50.0}
DECL FDAT FP286={TOOL_NO 2,BASE_NO 10,IPO_FRAME #BASE,POINT2[] " ",TQ_STATE FALSE}
DECL E6POS XP286={X 5.820,Y -6.990,Z 1.100,A 0.000,B 0.000,C -0.000}
DECL LDAT LCPDATC287={VEL 0.1,ACC 100,APO_DIST 5,APO_FAC 50.0,ORI_TYP #VAR,CIRC_TYP #BASE,JERK_FAC 50.0}
DECL FDAT FC287={TOOL_NO 2,BASE_NO 10,IPO_FRAME #BASE,POINT2[] " ",TQ_STATE FALSE}
DECL E6POS XCAux287={X -55.000,Y 5.930,Z 1.100,A 0.000,B 0.000,C -0.000}
DECL E6POS XCDes287={X -115.820,Y -6.990,Z 1.100,A 0.000,B 0.000,C -0.000}
DECL LDAT LCPDATC288={VEL 0.5,ACC 100,APO_DIST 5,APO_FAC 50.0,ORI_TYP #VAR,CIRC_TYP #BASE,JERK_FAC 50.0}
DECL FDAT FC288={TOOL_NO 2,BASE_NO 10,IPO_FRAME #BASE,POINT2[] " ",TQ_STATE FALSE}
DECL E6POS XCAux288={X -138.620,Y -19.630,Z 1.100,A 0.000,B 0.000,C -0.000}
DECL E6POS XCDes288={X -139.740,Y -17.970,Z 1.100,A 0.000,B 0.000,C -0.000}
DECL LDAT LCPDATP289={VEL 0.1,ACC 100,APO_DIST 5,APO_FAC 50.0,ORI_TYP #VAR,CIRC_TYP #BASE,JERK_FAC 50.0}
DECL FDAT FP289={TOOL_NO 2,BASE_NO 10,IPO_FRAME #BASE,POINT2[] " ",TQ_STATE FALSE}
DECL E6POS XP289={X -116.630,Y -5.170,Z 1.100,A 0.000,B 0.000,C -0.000}
DECL LDAT LCPDATC290={VEL 0.1,ACC 100,APO_DIST 5,APO_FAC 50.0,ORI_TYP #VAR,CIRC_TYP #BASE,JERK_FAC 50.0}
DECL FDAT FC290={TOOL_NO 2,BASE_NO 10,IPO_FRAME #BASE,POINT2[] " ",TQ_STATE FALSE}
DECL E6POS XCAux290={X -55.000,Y 7.930,Z 1.100,A 0.000,B 0.000,C -0.000}
DECL E6POS XCDes290={X 6.630,Y -5.170,Z 1.100,A 0.000,B 0.000,C -0.000}
DECL LDAT LCPDATC291={VEL 0.5,ACC 100,APO_DIST 5,APO_FAC 50.0,ORI_TYP #VAR,CIRC_TYP #BASE,JERK_FAC 50.0}
DECL FDAT FC291={TOOL_NO 2,BASE_NO 10,IPO_FRAME #BASE,POINT2[] " ",TQ_STATE FALSE}
DECL E6POS XCAux291={X 29.740,Y -17.970,Z 1.100,A 0.000,B 0.000,C -0.000}
DECL E6POS XCDes291={X 30.860,Y -16.310,Z 1.100,A 0.000,B 0.000,C -0.000}
DECL LDAT LCPDATP292={VEL 0.1,ACC 100,APO_DIST 5,APO_FAC 50.0,ORI_TYP #VAR,CIRC_TYP #BASE,JERK_FAC 50.0}
DECL FDAT FP292={TOOL_NO 2,BASE_NO 10,IPO_FRAME #BASE,POINT2[] " ",TQ_STATE FALSE}
DECL E6POS XP292={X 7.450,Y -3.340,Z 1.100,A 0.000,B 0.000,C -0.000}
DECL LDAT LCPDATC293={VEL 0.1,ACC 100,APO_DIST 5,APO_FAC 50.0,ORI_TYP #VAR,CIRC_TYP #BASE,JERK_FAC 50.0}
DECL FDAT FC293={TOOL_NO 2,BASE_NO 10,IPO_FRAME #BASE,POINT2[] " ",TQ_STATE FALSE}
DECL E6POS XCAux293={X -55.000,Y 9.930,Z 1.100,A 0.000,B 0.000,C -0.000}
DECL E6POS XCDes293={X -117.450,Y -3.340,Z 1.100,A 0.000,B 0.000,C -0.000}
DECL LDAT LCPDATC294={VEL 0.5,ACC 100,APO_DIST 5,APO_FAC 50.0,ORI_TYP #VAR,CIRC_TYP #BASE,JERK_FAC 50.0}
DECL FDAT FC294={TOOL_NO 2,BASE_NO 10,IPO_FRAME #BASE,POINT2[] " ",TQ_STATE FALSE}
DECL E6POS XCAux294={X -140.860,Y -16.310,Z 1.100,A 0.000,B 0.000,C -0.000}
DECL E6POS XCDes294={X -140.840,Y -16.330,Z 0.970,A -0.000,B -6.740,C -10.090}
DECL LDAT LCPDATP295={VEL 0.1,ACC 100,APO_DIST 5,APO_FAC 50.0,ORI_TYP #VAR,CIRC_TYP #BASE,JERK_FAC 50.0}
DECL FDAT FP295={TOOL_NO 2,BASE_NO 10,IPO_FRAME #BASE,POINT2[] " ",TQ_STATE FALSE}
DECL E6POS XP295={X -117.440,Y -3.360,Z 0.970,A -0.000,B -4.900,C -11.090}
DECL LDAT LCPDATC296={VEL 0.1,ACC 100,APO_DIST 5,APO_FAC 50.0,ORI_TYP #VAR,CIRC_TYP #BASE,JERK_FAC 50.0}
DECL FDAT FC296={TOOL_NO 2,BASE_NO 10,IPO_FRAME #BASE,POINT2[] " ",TQ_STATE FALSE}
DECL E6POS XCAux296={X -55.000,Y 9.910,Z 0.970,A 0.000,B 0.000,C -12.110}
DECL E6POS XCDes296={X 7.440,Y -3.360,Z 0.970,A 0.000,B 4.900,C -11.090}
DECL LDAT LCPDATC297={VEL 0.5,ACC 100,APO_DIST 5,APO_FAC 50.0,ORI_TYP #VAR,CIRC_TYP #BASE,JERK_FAC 50.0}
DECL FDAT FC297={TOOL_NO 2,BASE_NO 10,IPO_FRAME #BASE,POINT2[] " ",TQ_STATE FALSE}
DECL E6POS XCAux297={X 30.840,Y -16.330,Z 0.970,A 0.000,B 6.740,C -10.090}
DECL E6POS XCDes297={X 30.730,Y -16.500,Z 0.700,A 0.000,B 0.000,C -0.000}
DECL LDAT LCPDATP298={VEL 0.1,ACC 100,APO_DIST 5,APO_FAC 50.0,ORI_TYP #VAR,CIRC_TYP #BASE,JERK_FAC 50.0}
DECL FDAT FP298={TOOL_NO 2,BASE_NO 10,IPO_FRAME #BASE,POINT2[] " ",TQ_STATE FALSE}
DECL E6POS XP298={X 7.360,Y -3.540,Z 0.700,A 0.000,B 0.000,C -0.000}
DECL LDAT LCPDATC299={VEL 0.1,ACC 100,APO_DIST 5,APO_FAC 50.0,ORI_TYP #VAR,CIRC_TYP #BASE,JERK_FAC 50.0}
DECL FDAT FC299={TOOL_NO 2,BASE_NO 10,IPO_FRAME #BASE,POINT2[] " ",TQ_STATE FALSE}
DECL E6POS XCAux299={X -55.000,Y 9.710,Z 0.700,A 0.000,B 0.000,C -0.000}
DECL E6POS XCDes299={X -117.360,Y -3.540,Z 0.700,A 0.000,B 0.000,C -0.000}
DECL LDAT LCPDATC300={VEL 0.5,ACC 100,APO_DIST 5,APO_FAC 50.0,ORI_TYP #VAR,CIRC_TYP #BASE,JERK_FAC 50.0}
DECL FDAT FC300={TOOL_NO 2,BASE_NO 10,IPO_FRAME #BASE,POINT2[] " ",TQ_STATE FALSE}
DECL E6POS XCAux300={X -140.730,Y -16.500,Z 0.700,A 0.000,B 0.000,C -0.000}
DECL E6POS XCDes300={X -139.610,Y -18.160,Z 0.700,A 0.000,B 0.000,C -0.000}
DECL LDAT LCPDATP301={VEL 0.1,ACC 100,APO_DIST 5,APO_FAC 50.0,ORI_TYP #VAR,CIRC_TYP #BASE,JERK_FAC 50.0}
DECL FDAT FP301={TOOL_NO 2,BASE_NO 10,IPO_FRAME #BASE,POINT2[] " ",TQ_STATE FALSE}
DECL E6POS XP301={X -116.540,Y -5.370,Z 0.700,A 0.000,B 0.000,C -0.000}
DECL LDAT LCPDATC302={VEL 0.1,ACC 100,APO_DIST 5,APO_FAC 50.0,ORI_TYP #VAR,CIRC_TYP #BASE,JERK_FAC 50.0}
DECL FDAT FC302={TOOL_NO 2,BASE_NO 10,IPO_FRAME #BASE,POINT2[] " ",TQ_STATE FALSE}
DECL E6POS XCAux302={X -55.000,Y 7.710,Z 0.700,A 0.000,B 0.000,C -0.000}
DECL E6POS XCDes302={X 6.540,Y -5.370,Z 0.700,A 0.000,B 0.000,C -0.000}
DECL LDAT LCPDATC303={VEL 0.5,ACC 100,APO_DIST 5,APO_FAC 50.0,ORI_TYP #VAR,CIRC_TYP #BASE,JERK_FAC 50.0}
DECL FDAT FC303={TOOL_NO 2,BASE_NO 10,IPO_FRAME #BASE,POINT2[] " ",TQ_STATE FALSE}
DECL E6POS XCAux303={X 29.610,Y -18.160,Z 0.700,A 0.000,B 0.000,C -0.000}
DECL E6POS XCDes303={X 28.500,Y -19.810,Z 0.700,A 0.000,B 0.000,C -0.000}
DECL LDAT LCPDATP304={VEL 0.1,ACC 100,APO_DIST 5,APO_FAC 50.0,ORI_TYP #VAR,CIRC_TYP #BASE,JERK_FAC 50.0}
DECL FDAT FP304={TOOL_NO 2,BASE_NO 10,IPO_FRAME #BASE,POINT2[] " ",TQ_STATE FALSE}
DECL E6POS XP304={X 5.730,Y -7.200,Z 0.700,A 0.000,B 0.000,C -0.000}
DECL LDAT LCPDATC305={VEL 0.1,ACC 100,APO_DIST 5,APO_FAC 50.0,ORI_TYP #VAR,CIRC_TYP #BASE,JERK_FAC 50.0}
DECL FDAT FC305={TOOL_NO 2,BASE_NO 10,IPO_FRAME #BASE,POINT2[] " ",TQ_STATE FALSE}
DECL E6POS XCAux305={X -55.000,Y 5.710,Z 0.700,A 0.000,B 0.000,C -0.000}
DECL E6POS XCDes305={X -115.730,Y -7.200,Z 0.700,A 0.000,B 0.000,C -0.000}
DECL LDAT LCPDATC306={VEL 0.5,ACC 100,APO_DIST 5,APO_FAC 50.0,ORI_TYP #VAR,CIRC_TYP #BASE,JERK_FAC 50.0}
DECL FDAT FC306={TOOL_NO 2,BASE_NO 10,IPO_FRAME #BASE,POINT2[] " ",TQ_STATE FALSE}
DECL E6POS XCAux306={X -138.500,Y -19.810,Z 0.700,A 0.000,B 0.000,C -0.000}
DECL E6POS XCDes306={X -137.380,Y -21.470,Z 0.700,A 0.000,B 0.000,C -0.000}
DECL LDAT LCPDATP307={VEL 0.1,ACC 100,APO_DIST 5,APO_FAC 50.0,ORI_TYP #VAR,CIRC_TYP #BASE,JERK_FAC 50.0}
DECL FDAT FP307={TOOL_NO 2,BASE_NO 10,IPO_FRAME #BASE,POINT2[] " ",TQ_STATE FALSE}
DECL E6POS XP307={X -114.920,Y -9.020,Z 0.700,A 0.000,B 0.000,C -0.000}
DECL LDAT LCPDATC308={VEL 0.1,ACC 100,APO_DIST 5,APO_FAC 50.0,ORI_TYP #VAR,CIRC_TYP #BASE,JERK_FAC 50.0}
DECL FDAT FC308={TOOL_NO 2,BASE_NO 10,IPO_FRAME #BASE,POINT2[] " ",TQ_STATE FALSE}
DECL E6POS XCAux308={X -55.000,Y 3.710,Z 0.700,A 0.000,B 0.000,C -0.000}
DECL E6POS XCDes308={X 4.920,Y -9.020,Z 0.700,A 0.000,B 0.000,C -0.000}
DECL LDAT LCPDATC309={VEL 0.5,ACC 100,APO_DIST 5,APO_FAC 50.0,ORI_TYP #VAR,CIRC_TYP #BASE,JERK_FAC 50.0}
DECL FDAT FC309={TOOL_NO 2,BASE_NO 10,IPO_FRAME #BASE,POINT2[] " ",TQ_STATE FALSE}
DECL E6POS XCAux309={X 27.380,Y -21.470,Z 0.700,A 0.000,B 0.000,C -0.000}
DECL E6POS XCDes309={X 26.260,Y -23.130,Z 0.700,A 0.000,B 0.000,C -0.000}
DECL LDAT LCPDATP310={VEL 0.1,ACC 100,APO_DIST 5,APO_FAC 50.0,ORI_TYP #VAR,CIRC_TYP #BASE,JERK_FAC 50.0}
DECL FDAT FP310={TOOL_NO 2,BASE_NO 10,IPO_FRAME #BASE,POINT2[] " ",TQ_STATE FALSE}
DECL E6POS XP310={X 4.100,Y -10.850,Z 0.700,A 0.000,B 0.000,C -0.000}
DECL LDAT LCPDATC311={VEL 0.1,ACC 100,APO_DIST 5,APO_FAC 50.0,ORI_TYP #VAR,CIRC_TYP #BASE,JERK_FAC 50.0}
DECL FDAT FC311={TOOL_NO 2,BASE_NO 10,IPO_FRAME #BASE,POINT2[] " ",TQ_STATE FALSE}
DECL E6POS XCAux311={X -55.000,Y 1.710,Z 0.700,A 0.000,B 0.000,C -0.000}
DECL E6POS XCDes311={X -114.100,Y -10.850,Z 0.700,A 0.000,B 0.000,C -0.000}
DECL LDAT LCPDATC312={VEL 0.5,ACC 100,APO_DIST 5,APO_FAC 50.0,ORI_TYP #VAR,CIRC_TYP #BASE,JERK_FAC 50.0}
DECL FDAT FC312={TOOL_NO 2,BASE_NO 10,IPO_FRAME #BASE,POINT2[] " ",TQ_STATE FALSE}
DECL E6POS XCAux312={X -136.260,Y -23.130,Z 0.700,A 0.000,B 0.000,C -0.000}
DECL E6POS XCDes312={X -135.140,Y -24.790,Z 0.700,A 0.000,B 0.000,C -0.000}
DECL LDAT LCPDATP313={VEL 0.1,ACC 100,APO_DIST 5,APO_FAC 50.0,ORI_TYP #VAR,CIRC_TYP #BASE,JERK_FAC 50.0}
DECL FDAT FP313={TOOL_NO 2,BASE_NO 10,IPO_FRAME #BASE,POINT2[] " ",TQ_STATE FALSE}
DECL E6POS XP313={X -113.290,Y -12.680,Z 0.700,A 0.000,B 0.000,C -0.000}
DECL LDAT LCPDATC314={VEL 0.1,ACC 100,APO_DIST 5,APO_FAC 50.0,ORI_TYP #VAR,CIRC_TYP #BASE,JERK_FAC 50.0}
DECL FDAT FC314={TOOL_NO 2,BASE_NO 10,IPO_FRAME #BASE,POINT2[] " ",TQ_STATE FALSE}
DECL E6POS XCAux314={X -55.000,Y -0.290,Z 0.700,A 0.000,B 0.000,C -0.000}
DECL E6POS XCDes314={X 3.290,Y -12.680,Z 0.700,A 0.000,B 0.000,C -0.000}
DECL LDAT LCPDATC315={VEL 0.5,ACC 100,APO_DIST 5,APO_FAC 50.0,ORI_TYP #VAR,CIRC_TYP #BASE,JERK_FAC 50.0}
DECL FDAT FC315={TOOL_NO 2,BASE_NO 10,IPO_FRAME #BASE,POINT2[] " ",TQ_STATE FALSE}
DECL E6POS XCAux315={X 25.140,Y -24.790,Z 0.700,A 0.000,B 0.000,C -0.000}
DECL E6POS XCDes315={X 24.020,Y -26.450,Z 0.700,A 0.000,B 0.000,C -0.000}
DECL LDAT LCPDATP316={VEL 0.1,ACC 100,APO_DIST 5,APO_FAC 50.0,ORI_TYP #VAR,CIRC_TYP #BASE,JERK_FAC 50.0}
DECL FDAT FP316={TOOL_NO 2,BASE_NO 10,IPO_FRAME #BASE,POINT2[] " ",TQ_STATE FALSE}
DECL E6POS XP316={X 2.480,Y -14.500,Z 0.700,A 0.000,B 0.000,C -0.000}
DECL LDAT LCPDATC317={VEL 0.1,ACC 100,APO_DIST 5,APO_FAC 50.0,ORI_TYP #VAR,CIRC_TYP #BASE,JERK_FAC 50.0}
DECL FDAT FC317={TOOL_NO 2,BASE_NO 10,IPO_FRAME #BASE,POINT2[] " ",TQ_STATE FALSE}
DECL E6POS XCAux317={X -55.000,Y -2.290,Z 0.700,A 0.000,B 0.000,C -0.000}
DECL E6POS XCDes317={X -112.480,Y -14.500,Z 0.700,A 0.000,B 0.000,C -0.000}
DECL LDAT LCPDATC318={VEL 0.5,ACC 100,APO_DIST 5,APO_FAC 50.0,ORI_TYP #VAR,CIRC_TYP #BASE,JERK_FAC 50.0}
DECL FDAT FC318={TOOL_NO 2,BASE_NO 10,IPO_FRAME #BASE,POINT2[] " ",TQ_STATE FALSE}
DECL E6POS XCAux318={X -134.020,Y -26.450,Z 0.700,A 0.000,B 0.000,C -0.000}
DECL E6POS XCDes318={X -132.900,Y -28.100,Z 0.700,A 0.000,B 0.000,C -0.000}
DECL LDAT LCPDATP319={VEL 0.1,ACC 100,APO_DIST 5,APO_FAC 50.0,ORI_TYP #VAR,CIRC_TYP #BASE,JERK_FAC 50.0}
DECL FDAT FP319={TOOL_NO 2,BASE_NO 10,IPO_FRAME #BASE,POINT2[] " ",TQ_STATE FALSE}
DECL E6POS XP319={X -111.660,Y -16.330,Z 0.700,A 0.000,B 0.000,C -0.000}
DECL LDAT LCPDATC320={VEL 0.1,ACC 100,APO_DIST 5,APO_FAC 50.0,ORI_TYP #VAR,CIRC_TYP #BASE,JERK_FAC 50.0}
DECL FDAT FC320={TOOL_NO 2,BASE_NO 10,IPO_FRAME #BASE,POINT2[] " ",TQ_STATE FALSE}
